KUKA KRL program: f1_Kuka_APT207T02S07.SRC

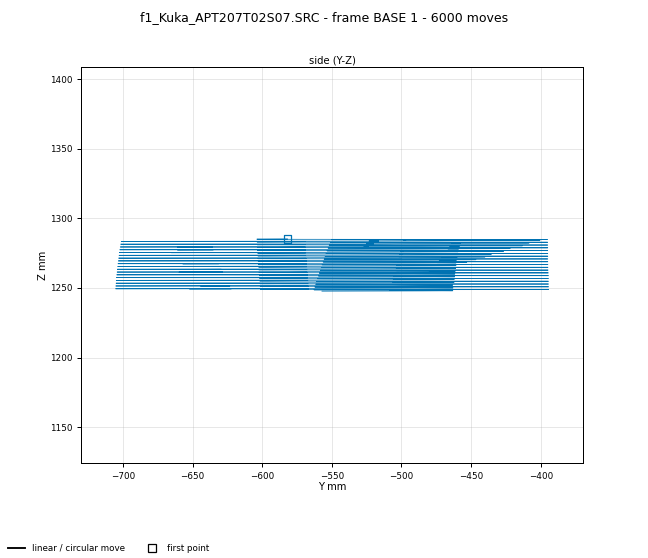
[picture p0: tool path of f1_Kuka_APT207T02S07.SRC in frame BASE 1, 6000 of 6001 moves have a stored position in this frame; points joined in program order, loops and branches not executed]
&ACCESS RVP
&REL 2
&PARAM TEMPLATE = C:\KRC\Roboter\Template\vorgabe
&PARAM EDITMASK = *
DEF f1_Kuka_APT207T02S07()


;FOLD INI;%{PE}%V3.2.0,%MKUKATPBASIS,%CINIT,%VCOMMON,%P
  ;FOLD BAS INI;%{E}%V3.2.0,%MKUKATPBASIS,%CINIT,%VINIT,%P
    GLOBAL INTERRUPT DECL 3 WHEN $STOPMESS==TRUE DO IR_STOPM ( )
    INTERRUPT ON 3
    BAS (#INITMOV,0 )
  ;ENDFOLD (BAS INI)
  ;FOLD USER INI;%{E}%V3.2.0,%MKUKATPUSER,%CINIT,%VINIT,%P
    ;Make your modifications here
  ;ENDFOLD (USER INI)
;ENDFOLD (INI)


;*** Make Null PTP Move
  PTP $pos_act

;*** Auto Load The Correct TOOL Data
  $tool=tool_data[2]

;*** Auto Load The Correct BASE Data
  $base=base_data[1]

  $ADVANCE = 5

;*** Restate Last Velocity
MMPM(30000.0)
SetRPM(8000)
LIN {X 0.048,Y -581.826,Z 1285.220,A 0.000,B 0.000,C 90.000,E1 75.589} C_DIS
LIN {X -0.200,Y -582.772,Z 1285.213,A 0.000,B 0.000,C 90.000,E1 74.267} C_DIS
LIN {X 0.309,Y -583.459,Z 1285.207,A 0.000,B 0.000,C 90.000,E1 73.142} C_DIS
LIN {X 0.170,Y -584.748,Z 1285.196,A 0.000,B 0.000,C 90.000,E1 71.275} C_DIS
LIN {X 0.250,Y -585.720,Z 1285.186,A 0.000,B 0.000,C 90.000,E1 69.390} C_DIS
LIN {X 0.080,Y -587.159,Z 1285.172,A 0.000,B 0.000,C 90.000,E1 66.997} C_DIS
LIN {X -0.086,Y -588.355,Z 1285.163,A 0.000,B 0.000,C 90.000,E1 65.409} C_DIS
LIN {X 0.318,Y -589.579,Z 1285.155,A 0.000,B 0.000,C 90.000,E1 63.768} C_DIS
LIN {X -0.318,Y -590.924,Z 1285.146,A 0.000,B 0.000,C 90.000,E1 62.231} C_DIS
LIN {X 0.047,Y -592.714,Z 1285.135,A 0.000,B 0.000,C 90.000,E1 60.333} C_DIS
LIN {X 0.246,Y -594.610,Z 1285.125,A 0.000,B 0.000,C 90.000,E1 58.456} C_DIS
LIN {X -0.011,Y -596.580,Z 1285.115,A 0.000,B 0.000,C 90.000,E1 56.628} C_DIS
LIN {X -0.137,Y -598.137,Z 1285.106,A 0.000,B 0.000,C 90.000,E1 55.055} C_DIS
LIN {X -0.029,Y -599.606,Z 1285.097,A 0.000,B 0.000,C 90.000,E1 53.463} C_DIS
LIN {X -0.243,Y -600.936,Z 1285.088,A 0.000,B 0.000,C 90.000,E1 51.904} C_DIS
LIN {X 0.057,Y -601.935,Z 1285.081,A 0.000,B 0.000,C 90.000,E1 50.561} C_DIS
LIN {X -0.015,Y -602.640,Z 1285.074,A 0.000,B 0.000,C 90.000,E1 49.256} C_DIS
LIN {X 0.252,Y -603.219,Z 1285.066,A 0.000,B 0.000,C 90.000,E1 47.919} C_DIS
LIN {X 0.129,Y -603.619,Z 1285.059,A 0.000,B 0.000,C 90.000,E1 46.620} C_DIS
LIN {X 0.184,Y -603.812,Z 1285.053,A 0.000,B 0.000,C 90.000,E1 45.567} C_DIS
LIN {X 0.047,Y -603.766,Z 1285.046,A 0.000,B 0.000,C 90.000,E1 44.271} C_DIS
LIN {X 0.303,Y -603.652,Z 1285.042,A 0.000,B 0.000,C 90.000,E1 43.461} C_DIS
LIN {X -0.019,Y -603.203,Z 1285.033,A 0.000,B 0.000,C 90.000,E1 41.919} C_DIS
LIN {X -0.182,Y -602.884,Z 1285.029,A 0.000,B 0.000,C 90.000,E1 41.148} C_DIS
LIN {X 0.183,Y -602.034,Z 1285.018,A 0.000,B 0.000,C 90.000,E1 39.277} C_DIS
LIN {X -0.130,Y -601.379,Z 1285.013,A 0.000,B 0.000,C 90.000,E1 38.257} C_DIS
LIN {X -0.203,Y -600.134,Z 1285.005,A 0.000,B 0.000,C 90.000,E1 36.950} C_DIS
LIN {X 0.177,Y -598.525,Z 1284.998,A 0.000,B 0.000,C 90.000,E1 35.598} C_DIS
LIN {X 0.054,Y -597.309,Z 1284.994,A 0.000,B 0.000,C 90.000,E1 34.818} C_DIS
LIN {X -0.084,Y -595.954,Z 1284.989,A 0.000,B 0.000,C 90.000,E1 34.040} C_DIS
LIN {X 0.147,Y -593.900,Z 1284.983,A 0.000,B 0.000,C 90.000,E1 32.959} C_DIS
LIN {X 0.253,Y -592.666,Z 1284.980,A 0.000,B 0.000,C 90.000,E1 32.418} C_DIS
LIN {X -0.062,Y -589.778,Z 1284.974,A 0.000,B 0.000,C 90.000,E1 31.386} C_DIS
LIN {X 0.014,Y -588.135,Z 1284.971,A 0.000,B 0.000,C 90.000,E1 30.846} C_DIS
LIN {X -0.045,Y -585.442,Z 1284.967,A 0.000,B 0.000,C 90.000,E1 30.050} C_DIS
LIN {X 0.376,Y -582.311,Z 1284.963,A 0.000,B 0.000,C 90.000,E1 29.205} C_DIS
LIN {X 0.046,Y -579.263,Z 1284.959,A 0.000,B 0.000,C 90.000,E1 28.565} C_DIS
LIN {X -0.185,Y -574.540,Z 1284.953,A 0.000,B 0.000,C 90.000,E1 27.641} C_DIS
LIN {X -0.067,Y -570.770,Z 1284.950,A 0.000,B 0.000,C 90.000,E1 26.950} C_DIS
LIN {X 0.275,Y -566.596,Z 1284.946,A 0.000,B 0.000,C 90.000,E1 26.232} C_DIS
LIN {X -0.088,Y -563.016,Z 1284.943,A 0.000,B 0.000,C 90.000,E1 25.720} C_DIS
LIN {X -0.067,Y -558.285,Z 1284.939,A 0.000,B 0.000,C 90.000,E1 25.027} C_DIS
LIN {X -0.011,Y -553.284,Z 1284.935,A 0.000,B 0.000,C 90.000,E1 24.335} C_DIS
LIN {X 0.041,Y -548.855,Z 1284.932,A 0.000,B 0.000,C 90.000,E1 23.770} C_DIS
LIN {X 0.218,Y -540.504,Z 1284.927,A 0.000,B 0.000,C 90.000,E1 22.770} C_DIS
LIN {X 0.093,Y -534.167,Z 1284.923,A 0.000,B 0.000,C 90.000,E1 22.078} C_DIS
LIN {X 0.176,Y -526.388,Z 1284.918,A 0.000,B 0.000,C 90.000,E1 21.227} C_DIS
LIN {X 0.260,Y -515.939,Z 1284.912,A 0.000,B 0.000,C 90.000,E1 20.120} C_DIS
LIN {X 0.127,Y -503.629,Z 1284.905,A 0.000,B 0.000,C 90.000,E1 18.906} C_DIS
LIN {X -0.214,Y -493.980,Z 1284.900,A 0.000,B 0.000,C 90.000,E1 18.000} C_DIS
LIN {X 0.123,Y -485.479,Z 1284.896,A 0.000,B 0.000,C 90.000,E1 17.166} C_DIS
LIN {X -0.200,Y -477.046,Z 1284.891,A 0.000,B 0.000,C 90.000,E1 16.441} C_DIS
LIN {X 0.098,Y -466.700,Z 1284.886,A 0.000,B 0.000,C 90.000,E1 15.481} C_DIS
LIN {X 0.071,Y -446.110,Z 1284.876,A 0.000,B 0.000,C 90.000,E1 13.592} C_DIS
LIN {X -0.108,Y -422.917,Z 1284.863,A 0.000,B 0.000,C 90.000,E1 11.299} C_DIS
LIN {X -0.089,Y -405.684,Z 1284.852,A 0.000,B 0.000,C 90.000,E1 9.434} C_DIS
LIN {X -0.183,Y -400.098,Z 1284.849,A 0.000,B 0.000,C 90.000,E1 8.803} C_DIS
LIN {X 0.108,Y -396.550,Z 1284.846,A 0.000,B 0.000,C 90.000,E1 8.276} C_DIS
LIN {X -0.073,Y -395.161,Z 1284.845,A 0.000,B 0.000,C 90.000,E1 8.049} C_DIS
LIN {X -0.110,Y -395.161,Z 1284.845,A 0.000,B 0.000,C 90.000,E1 8.049} C_DIS
LIN {X 0.067,Y -395.273,Z 1284.844,A 0.000,B 0.000,C 90.000,E1 7.936} C_DIS
LIN {X 0.028,Y -395.301,Z 1284.844,A 0.000,B 0.000,C 90.000,E1 7.936} C_DIS
LIN {X 0.134,Y -395.933,Z 1284.844,A 0.000,B 0.000,C 90.000,E1 7.814} C_DIS
LIN {X 0.006,Y -399.237,Z 1284.842,A 0.000,B 0.000,C 90.000,E1 7.530} C_DIS
LIN {X 0.124,Y -403.414,Z 1284.840,A 0.000,B 0.000,C 90.000,E1 7.239} C_DIS
LIN {X 0.177,Y -410.405,Z 1284.838,A 0.000,B 0.000,C 90.000,E1 6.834} C_DIS
LIN {X 0.174,Y -416.754,Z 1284.836,A 0.000,B 0.000,C 90.000,E1 6.429} C_DIS
LIN {X -0.121,Y -423.072,Z 1284.833,A 0.000,B 0.000,C 90.000,E1 6.024} C_DIS
LIN {X -0.122,Y -430.624,Z 1284.830,A 0.000,B 0.000,C 90.000,E1 5.448} C_DIS
LIN {X -0.194,Y -441.583,Z 1284.825,A 0.000,B 0.000,C 90.000,E1 4.588} C_DIS
LIN {X -0.037,Y -452.155,Z 1284.820,A 0.000,B 0.000,C 90.000,E1 3.669} C_DIS
LIN {X 0.164,Y -459.533,Z 1284.817,A 0.000,B 0.000,C 90.000,E1 2.980} C_DIS
LIN {X 0.220,Y -466.501,Z 1284.813,A 0.000,B 0.000,C 90.000,E1 2.293} C_DIS
LIN {X -0.131,Y -473.329,Z 1284.809,A 0.000,B 0.000,C 90.000,E1 1.604} C_DIS
LIN {X 0.114,Y -478.651,Z 1284.806,A 0.000,B 0.000,C 90.000,E1 0.974} C_DIS
LIN {X -0.058,Y -484.810,Z 1284.801,A 0.000,B 0.000,C 90.000,E1 0.229} C_DIS
LIN {X 0.015,Y -490.312,Z 1284.797,A 0.000,B 0.000,C 90.000,E1 359.484} C_DIS
LIN {X 0.044,Y -496.441,Z 1284.792,A 0.000,B 0.000,C 90.000,E1 358.568} C_DIS
LIN {X -0.029,Y -501.231,Z 1284.788,A 0.000,B 0.000,C 90.000,E1 357.822} C_DIS
LIN {X 0.231,Y -504.859,Z 1284.785,A 0.000,B 0.000,C 90.000,E1 357.192} C_DIS
LIN {X 0.241,Y -509.077,Z 1284.780,A 0.000,B 0.000,C 90.000,E1 356.445} C_DIS
LIN {X -0.218,Y -513.021,Z 1284.776,A 0.000,B 0.000,C 90.000,E1 355.755} C_DIS
LIN {X -0.210,Y -518.124,Z 1284.771,A 0.000,B 0.000,C 90.000,E1 354.723} C_DIS
LIN {X -0.090,Y -522.655,Z 1284.765,A 0.000,B 0.000,C 90.000,E1 353.685} C_DIS
LIN {X 0.087,Y -526.892,Z 1284.759,A 0.000,B 0.000,C 90.000,E1 352.648} C_DIS
LIN {X 0.101,Y -531.063,Z 1284.753,A 0.000,B 0.000,C 90.000,E1 351.489} C_DIS
LIN {X 0.130,Y -533.929,Z 1284.748,A 0.000,B 0.000,C 90.000,E1 350.622} C_DIS
LIN {X -0.250,Y -536.492,Z 1284.743,A 0.000,B 0.000,C 90.000,E1 349.803} C_DIS
LIN {X -0.069,Y -538.784,Z 1284.739,A 0.000,B 0.000,C 90.000,E1 348.926} C_DIS
LIN {X 0.214,Y -541.529,Z 1284.732,A 0.000,B 0.000,C 90.000,E1 347.757} C_DIS
LIN {X 0.003,Y -543.947,Z 1284.726,A 0.000,B 0.000,C 90.000,E1 346.645} C_DIS
LIN {X 0.172,Y -545.083,Z 1284.723,A 0.000,B 0.000,C 90.000,E1 346.061} C_DIS
LIN {X 0.131,Y -546.942,Z 1284.716,A 0.000,B 0.000,C 90.000,E1 344.936} C_DIS
LIN {X 0.021,Y -548.089,Z 1284.712,A 0.000,B 0.000,C 90.000,E1 344.102} C_DIS
LIN {X -0.075,Y -548.968,Z 1284.707,A 0.000,B 0.000,C 90.000,E1 343.268} C_DIS
LIN {X 0.091,Y -549.899,Z 1284.701,A 0.000,B 0.000,C 90.000,E1 342.127} C_DIS
LIN {X 0.182,Y -550.312,Z 1284.696,A 0.000,B 0.000,C 90.000,E1 341.275} C_DIS
LIN {X 0.280,Y -550.335,Z 1284.691,A 0.000,B 0.000,C 90.000,E1 340.423} C_DIS
LIN {X -0.136,Y -550.059,Z 1284.687,A 0.000,B 0.000,C 90.000,E1 339.625} C_DIS
LIN {X 0.206,Y -549.736,Z 1284.684,A 0.000,B 0.000,C 90.000,E1 339.028} C_DIS
LIN {X 0.227,Y -549.232,Z 1284.681,A 0.000,B 0.000,C 90.000,E1 338.465} C_DIS
LIN {X -0.202,Y -548.198,Z 1284.676,A 0.000,B 0.000,C 90.000,E1 337.667} C_DIS
LIN {X 0.074,Y -546.828,Z 1284.671,A 0.000,B 0.000,C 90.000,E1 336.794} C_DIS
LIN {X -0.164,Y -545.362,Z 1284.667,A 0.000,B 0.000,C 90.000,E1 335.973} C_DIS
LIN {X -0.165,Y -544.289,Z 1284.663,A 0.000,B 0.000,C 90.000,E1 335.409} C_DIS
LIN {X 0.086,Y -542.056,Z 1284.659,A 0.000,B 0.000,C 90.000,E1 334.537} C_DIS
LIN {X 0.033,Y -539.633,Z 1284.654,A 0.000,B 0.000,C 90.000,E1 333.691} C_DIS
LIN {X -0.283,Y -536.936,Z 1284.649,A 0.000,B 0.000,C 90.000,E1 332.871} C_DIS
LIN {X 0.089,Y -533.883,Z 1284.644,A 0.000,B 0.000,C 90.000,E1 331.975} C_DIS
LIN {X 0.243,Y -531.727,Z 1284.641,A 0.000,B 0.000,C 90.000,E1 331.385} C_DIS
LIN {X 0.231,Y -528.707,Z 1284.637,A 0.000,B 0.000,C 90.000,E1 330.667} C_DIS
LIN {X 0.293,Y -524.436,Z 1284.632,A 0.000,B 0.000,C 90.000,E1 329.793} C_DIS
LIN {X -0.076,Y -521.409,Z 1284.629,A 0.000,B 0.000,C 90.000,E1 329.253} C_DIS
LIN {X -0.168,Y -508.672,Z 1284.616,A 0.000,B 0.000,C 90.000,E1 326.914} C_DIS
LIN {X -0.044,Y -504.398,Z 1284.611,A 0.000,B 0.000,C 90.000,E1 326.008} C_DIS
LIN {X -0.108,Y -501.931,Z 1284.607,A 0.000,B 0.000,C 90.000,E1 325.308} C_DIS
LIN {X 0.189,Y -501.065,Z 1284.606,A 0.000,B 0.000,C 90.000,E1 324.975} C_DIS
LIN {X -0.063,Y -499.234,Z 1284.601,A 0.000,B 0.000,C 90.000,E1 324.116} C_DIS
LIN {X -0.038,Y -497.969,Z 1284.596,A 0.000,B 0.000,C 90.000,E1 323.210} C_DIS
LIN {X 0.136,Y -497.147,Z 1284.589,A 0.000,B 0.000,C 90.000,E1 321.984} C_DIS
LIN {X -0.229,Y -496.725,Z 1284.581,A 0.000,B 0.000,C 90.000,E1 320.517} C_DIS
LIN {X 0.043,Y -496.935,Z 1284.572,A 0.000,B 0.000,C 90.000,E1 318.976} C_DIS
LIN {X 0.039,Y -497.249,Z 1284.560,A 0.000,B 0.000,C 90.000,E1 316.863} C_DIS
LIN {X -0.207,Y -497.490,Z 1284.550,A 0.000,B 0.000,C 90.000,E1 315.081} C_DIS
LIN {X -0.203,Y -497.954,Z 1284.535,A 0.000,B 0.000,C 90.000,E1 312.366} C_DIS
LIN {X 0.091,Y -498.258,Z 1284.527,A 0.000,B 0.000,C 90.000,E1 310.825} C_DIS
LIN {X -0.122,Y -498.440,Z 1284.520,A 0.000,B 0.000,C 90.000,E1 309.644} C_DIS
LIN {X -0.199,Y -498.339,Z 1284.515,A 0.000,B 0.000,C 90.000,E1 308.749} C_DIS
LIN {X 0.112,Y -497.903,Z 1284.510,A 0.000,B 0.000,C 90.000,E1 307.810} C_DIS
LIN {X -0.148,Y -497.351,Z 1284.507,A 0.000,B 0.000,C 90.000,E1 307.237} C_DIS
LIN {X 0.284,Y -496.489,Z 1284.503,A 0.000,B 0.000,C 90.000,E1 306.583} C_DIS
LIN {X 0.151,Y -495.889,Z 1284.502,A 0.000,B 0.000,C 90.000,E1 306.297} C_DIS
LIN {X 0.015,Y -495.108,Z 1284.500,A 0.000,B 0.000,C 90.000,E1 306.011} C_DIS
LIN {X -0.122,Y -493.974,Z 1284.498,A 0.000,B 0.000,C 90.000,E1 305.724} C_DIS
LIN {X 0.004,Y -476.992,Z 1284.482,A 0.000,B 0.000,C 90.000,E1 302.801} C_DIS
LIN {X -0.163,Y -462.651,Z 1284.467,A 0.000,B 0.000,C 90.000,E1 300.001} C_DIS
LIN {X -0.075,Y -449.320,Z 1284.450,A 0.000,B 0.000,C 90.000,E1 296.950} C_DIS
LIN {X 0.022,Y -438.317,Z 1284.433,A 0.000,B 0.000,C 90.000,E1 294.003} C_DIS
LIN {X 0.060,Y -427.853,Z 1284.415,A 0.000,B 0.000,C 90.000,E1 290.684} C_DIS
LIN {X 0.007,Y -418.374,Z 1284.394,A 0.000,B 0.000,C 90.000,E1 286.985} C_DIS
LIN {X 0.007,Y -410.353,Z 1284.372,A 0.000,B 0.000,C 90.000,E1 282.883} C_DIS
LIN {X 0.108,Y -405.581,Z 1284.353,A 0.000,B 0.000,C 90.000,E1 279.500} C_DIS
LIN {X -0.078,Y -405.689,Z 1284.333,A 0.000,B 0.000,C 90.000,E1 275.967} C_DIS
LIN {X -0.040,Y -403.463,Z 1284.304,A 0.000,B 0.000,C 90.000,E1 270.745} C_DIS
LIN {X -0.073,Y -403.247,Z 1284.302,A 0.000,B 0.000,C 90.000,E1 270.401} C_DIS
LIN {X 0.093,Y -400.475,Z 1284.286,A 0.000,B 0.000,C 90.000,E1 267.421} C_DIS
LIN {X 0.055,Y -400.476,Z 1284.286,A 0.000,B 0.000,C 90.000,E1 267.421} C_DIS
LIN {X -0.055,Y -405.330,Z 1284.250,A 0.000,B 0.000,C 90.000,E1 260.971} C_DIS
LIN {X 0.004,Y -411.969,Z 1284.225,A 0.000,B 0.000,C 90.000,E1 256.464} C_DIS
LIN {X -0.169,Y -419.748,Z 1284.204,A 0.000,B 0.000,C 90.000,E1 252.725} C_DIS
LIN {X -0.092,Y -428.611,Z 1284.185,A 0.000,B 0.000,C 90.000,E1 249.337} C_DIS
LIN {X 0.007,Y -439.259,Z 1284.167,A 0.000,B 0.000,C 90.000,E1 245.997} C_DIS
LIN {X 0.176,Y -451.103,Z 1284.149,A 0.000,B 0.000,C 90.000,E1 242.871} C_DIS
LIN {X 0.067,Y -460.165,Z 1284.138,A 0.000,B 0.000,C 90.000,E1 240.795} C_DIS
LIN {X 0.188,Y -461.036,Z 1284.136,A 0.000,B 0.000,C 90.000,E1 240.461} C_DIS
LIN {X -0.088,Y -461.611,Z 1284.134,A 0.000,B 0.000,C 90.000,E1 240.177} C_DIS
LIN {X -0.062,Y -462.296,Z 1284.131,A 0.000,B 0.000,C 90.000,E1 239.537} C_DIS
LIN {X 0.203,Y -462.605,Z 1284.127,A 0.000,B 0.000,C 90.000,E1 238.869} C_DIS
LIN {X -0.033,Y -462.663,Z 1284.122,A 0.000,B 0.000,C 90.000,E1 237.946} C_DIS
LIN {X -0.027,Y -462.349,Z 1284.117,A 0.000,B 0.000,C 90.000,E1 236.993} C_DIS
LIN {X -0.021,Y -461.709,Z 1284.110,A 0.000,B 0.000,C 90.000,E1 235.722} C_DIS
LIN {X -0.015,Y -460.306,Z 1284.095,A 0.000,B 0.000,C 90.000,E1 233.176} C_DIS
LIN {X 0.090,Y -459.422,Z 1284.085,A 0.000,B 0.000,C 90.000,E1 231.251} C_DIS
LIN {X 0.149,Y -458.484,Z 1284.071,A 0.000,B 0.000,C 90.000,E1 228.690} C_DIS
LIN {X 0.108,Y -457.814,Z 1284.058,A 0.000,B 0.000,C 90.000,E1 226.458} C_DIS
LIN {X -0.268,Y -457.345,Z 1284.044,A 0.000,B 0.000,C 90.000,E1 223.947} C_DIS
LIN {X 0.127,Y -457.909,Z 1284.024,A 0.000,B 0.000,C 90.000,E1 220.378} C_DIS
LIN {X -0.164,Y -458.661,Z 1284.012,A 0.000,B 0.000,C 90.000,E1 218.177} C_DIS
LIN {X 0.145,Y -463.330,Z 1283.978,A 0.000,B 0.000,C 90.000,E1 212.084} C_DIS
LIN {X 0.099,Y -466.009,Z 1283.966,A 0.000,B 0.000,C 90.000,E1 209.873} C_DIS
LIN {X -0.040,Y -469.420,Z 1283.950,A 0.000,B 0.000,C 90.000,E1 207.052} C_DIS
LIN {X 0.108,Y -471.545,Z 1283.942,A 0.000,B 0.000,C 90.000,E1 205.463} C_DIS
LIN {X 0.074,Y -474.369,Z 1283.931,A 0.000,B 0.000,C 90.000,E1 203.590} C_DIS
LIN {X 0.051,Y -478.675,Z 1283.916,A 0.000,B 0.000,C 90.000,E1 200.791} C_DIS
LIN {X 0.112,Y -482.749,Z 1283.902,A 0.000,B 0.000,C 90.000,E1 198.308} C_DIS
LIN {X -0.183,Y -485.961,Z 1283.892,A 0.000,B 0.000,C 90.000,E1 196.496} C_DIS
LIN {X -0.096,Y -488.690,Z 1283.883,A 0.000,B 0.000,C 90.000,E1 194.954} C_DIS
LIN {X 0.042,Y -491.381,Z 1283.875,A 0.000,B 0.000,C 90.000,E1 193.411} C_DIS
LIN {X 0.111,Y -494.109,Z 1283.866,A 0.000,B 0.000,C 90.000,E1 191.883} C_DIS
LIN {X 0.129,Y -496.849,Z 1283.858,A 0.000,B 0.000,C 90.000,E1 190.366} C_DIS
LIN {X -0.044,Y -500.740,Z 1283.846,A 0.000,B 0.000,C 90.000,E1 188.276} C_DIS
LIN {X 0.155,Y -502.380,Z 1283.841,A 0.000,B 0.000,C 90.000,E1 187.352} C_DIS
LIN {X -0.253,Y -504.575,Z 1283.834,A 0.000,B 0.000,C 90.000,E1 186.201} C_DIS
LIN {X -0.192,Y -507.140,Z 1283.826,A 0.000,B 0.000,C 90.000,E1 184.702} C_DIS
LIN {X -0.162,Y -509.747,Z 1283.818,A 0.000,B 0.000,C 90.000,E1 183.212} C_DIS
LIN {X -0.057,Y -512.196,Z 1283.810,A 0.000,B 0.000,C 90.000,E1 181.718} C_DIS
LIN {X 0.134,Y -514.028,Z 1283.803,A 0.000,B 0.000,C 90.000,E1 180.516} C_DIS
LIN {X -0.089,Y -515.367,Z 1283.798,A 0.000,B 0.000,C 90.000,E1 179.656} C_DIS
LIN {X 0.101,Y -517.474,Z 1283.790,A 0.000,B 0.000,C 90.000,E1 178.165} C_DIS
LIN {X -0.152,Y -518.982,Z 1283.783,A 0.000,B 0.000,C 90.000,E1 177.020} C_DIS
LIN {X 0.190,Y -520.307,Z 1283.777,A 0.000,B 0.000,C 90.000,E1 175.812} C_DIS
LIN {X -0.019,Y -521.600,Z 1283.769,A 0.000,B 0.000,C 90.000,E1 174.375} C_DIS
LIN {X -0.152,Y -522.343,Z 1283.762,A 0.000,B 0.000,C 90.000,E1 173.223} C_DIS
LIN {X -0.280,Y -523.033,Z 1283.754,A 0.000,B 0.000,C 90.000,E1 171.781} C_DIS
LIN {X 0.183,Y -523.263,Z 1283.748,A 0.000,B 0.000,C 90.000,E1 170.566} C_DIS
LIN {X 0.231,Y -523.185,Z 1283.740,A 0.000,B 0.000,C 90.000,E1 169.106} C_DIS
LIN {X -0.230,Y -522.561,Z 1283.732,A 0.000,B 0.000,C 90.000,E1 167.701} C_DIS
LIN {X -0.083,Y -521.708,Z 1283.725,A 0.000,B 0.000,C 90.000,E1 166.520} C_DIS
LIN {X 0.055,Y -520.793,Z 1283.719,A 0.000,B 0.000,C 90.000,E1 165.338} C_DIS
LIN {X -0.201,Y -519.262,Z 1283.709,A 0.000,B 0.000,C 90.000,E1 163.614} C_DIS
LIN {X 0.118,Y -517.420,Z 1283.698,A 0.000,B 0.000,C 90.000,E1 161.529} C_DIS
LIN {X -0.141,Y -516.682,Z 1283.693,A 0.000,B 0.000,C 90.000,E1 160.678} C_DIS
LIN {X -0.141,Y -516.324,Z 1283.684,A 0.000,B 0.000,C 90.000,E1 159.209} C_DIS
LIN {X 0.259,Y -516.711,Z 1283.680,A 0.000,B 0.000,C 90.000,E1 158.284} C_DIS
LIN {X 0.324,Y -517.764,Z 1283.673,A 0.000,B 0.000,C 90.000,E1 157.102} C_DIS
LIN {X 0.124,Y -518.879,Z 1283.670,A 0.000,B 0.000,C 90.000,E1 156.538} C_DIS
LIN {X -0.068,Y -520.301,Z 1283.667,A 0.000,B 0.000,C 90.000,E1 155.973} C_DIS
LIN {X 0.224,Y -522.225,Z 1283.663,A 0.000,B 0.000,C 90.000,E1 155.357} C_DIS
LIN {X 0.053,Y -524.712,Z 1283.660,A 0.000,B 0.000,C 90.000,E1 154.793} C_DIS
LIN {X -0.025,Y -528.710,Z 1283.656,A 0.000,B 0.000,C 90.000,E1 154.076} C_DIS
LIN {X -0.003,Y -531.578,Z 1283.654,A 0.000,B 0.000,C 90.000,E1 153.640} C_DIS
LIN {X -0.089,Y -539.433,Z 1283.648,A 0.000,B 0.000,C 90.000,E1 152.666} C_DIS
LIN {X 0.271,Y -548.357,Z 1283.643,A 0.000,B 0.000,C 90.000,E1 151.641} C_DIS
LIN {X 0.153,Y -565.525,Z 1283.633,A 0.000,B 0.000,C 90.000,E1 149.999} C_DIS
LIN {X -0.047,Y -574.734,Z 1283.629,A 0.000,B 0.000,C 90.000,E1 149.154} C_DIS
LIN {X -0.057,Y -581.132,Z 1283.625,A 0.000,B 0.000,C 90.000,E1 148.535} C_DIS
LIN {X -0.226,Y -589.974,Z 1283.620,A 0.000,B 0.000,C 90.000,E1 147.661} C_DIS
LIN {X -0.070,Y -596.134,Z 1283.617,A 0.000,B 0.000,C 90.000,E1 146.993} C_DIS
LIN {X -0.164,Y -601.805,Z 1283.613,A 0.000,B 0.000,C 90.000,E1 146.342} C_DIS
LIN {X -0.005,Y -606.058,Z 1283.610,A 0.000,B 0.000,C 90.000,E1 145.801} C_DIS
LIN {X 0.182,Y -610.024,Z 1283.607,A 0.000,B 0.000,C 90.000,E1 145.261} C_DIS
LIN {X 0.218,Y -614.724,Z 1283.604,A 0.000,B 0.000,C 90.000,E1 144.609} C_DIS
LIN {X -0.038,Y -618.124,Z 1283.601,A 0.000,B 0.000,C 90.000,E1 144.116} C_DIS
LIN {X 0.050,Y -622.762,Z 1283.596,A 0.000,B 0.000,C 90.000,E1 143.336} C_DIS
LIN {X -0.158,Y -625.657,Z 1283.594,A 0.000,B 0.000,C 90.000,E1 142.844} C_DIS
LIN {X 0.165,Y -627.743,Z 1283.591,A 0.000,B 0.000,C 90.000,E1 142.431} C_DIS
LIN {X 0.125,Y -633.916,Z 1283.584,A 0.000,B 0.000,C 90.000,E1 141.170} C_DIS
LIN {X -0.247,Y -638.218,Z 1283.579,A 0.000,B 0.000,C 90.000,E1 140.194} C_DIS
LIN {X -0.079,Y -642.231,Z 1283.573,A 0.000,B 0.000,C 90.000,E1 139.175} C_DIS
LIN {X 0.002,Y -646.873,Z 1283.566,A 0.000,B 0.000,C 90.000,E1 137.919} C_DIS
LIN {X 0.227,Y -650.332,Z 1283.561,A 0.000,B 0.000,C 90.000,E1 136.905} C_DIS
LIN {X -0.003,Y -654.618,Z 1283.554,A 0.000,B 0.000,C 90.000,E1 135.688} C_DIS
LIN {X 0.231,Y -660.564,Z 1283.544,A 0.000,B 0.000,C 90.000,E1 133.947} C_DIS
LIN {X -0.309,Y -664.882,Z 1283.537,A 0.000,B 0.000,C 90.000,E1 132.771} C_DIS
LIN {X 0.155,Y -669.089,Z 1283.531,A 0.000,B 0.000,C 90.000,E1 131.515} C_DIS
LIN {X -0.184,Y -673.808,Z 1283.523,A 0.000,B 0.000,C 90.000,E1 130.092} C_DIS
LIN {X -0.029,Y -677.602,Z 1283.516,A 0.000,B 0.000,C 90.000,E1 128.874} C_DIS
LIN {X -0.290,Y -679.747,Z 1283.512,A 0.000,B 0.000,C 90.000,E1 128.177} C_DIS
LIN {X 0.070,Y -683.148,Z 1283.505,A 0.000,B 0.000,C 90.000,E1 126.950} C_DIS
LIN {X 0.082,Y -686.305,Z 1283.499,A 0.000,B 0.000,C 90.000,E1 125.758} C_DIS
LIN {X -0.418,Y -689.158,Z 1283.492,A 0.000,B 0.000,C 90.000,E1 124.612} C_DIS
LIN {X 0.041,Y -691.302,Z 1283.487,A 0.000,B 0.000,C 90.000,E1 123.627} C_DIS
LIN {X 0.122,Y -692.680,Z 1283.483,A 0.000,B 0.000,C 90.000,E1 122.911} C_DIS
LIN {X -0.338,Y -694.452,Z 1283.478,A 0.000,B 0.000,C 90.000,E1 122.005} C_DIS
LIN {X 0.048,Y -696.407,Z 1283.471,A 0.000,B 0.000,C 90.000,E1 120.797} C_DIS
LIN {X -0.144,Y -697.875,Z 1283.466,A 0.000,B 0.000,C 90.000,E1 119.873} C_DIS
LIN {X -0.052,Y -699.481,Z 1283.459,A 0.000,B 0.000,C 90.000,E1 118.693} C_DIS
LIN {X -0.210,Y -700.493,Z 1283.454,A 0.000,B 0.000,C 90.000,E1 117.769} C_DIS
LIN {X -0.017,Y -701.034,Z 1283.450,A 0.000,B 0.000,C 90.000,E1 117.052} C_DIS
LIN {X 0.140,Y -701.210,Z 1283.445,A 0.000,B 0.000,C 90.000,E1 116.104} C_DIS
LIN {X -0.215,Y -701.232,Z 1283.444,A 0.000,B 0.000,C 90.000,E1 115.899} C_DIS
LIN {X 0.306,Y -700.865,Z 1283.440,A 0.000,B 0.000,C 90.000,E1 115.155} C_DIS
LIN {X -0.077,Y -700.397,Z 1283.437,A 0.000,B 0.000,C 90.000,E1 114.719} C_DIS
LIN {X -0.171,Y -699.673,Z 1283.435,A 0.000,B 0.000,C 90.000,E1 114.259} C_DIS
LIN {X -0.189,Y -699.008,Z 1283.433,A 0.000,B 0.000,C 90.000,E1 114.027} C_DIS
LIN {X 0.342,Y -697.245,Z 1283.431,A 0.000,B 0.000,C 90.000,E1 113.515} C_DIS
LIN {X -0.168,Y -696.536,Z 1283.430,A 0.000,B 0.000,C 90.000,E1 113.439} C_DIS
LIN {X 0.062,Y -693.012,Z 1283.428,A 0.000,B 0.000,C 90.000,E1 112.950} C_DIS
LIN {X 0.185,Y -691.812,Z 1283.427,A 0.000,B 0.000,C 90.000,E1 112.823} C_DIS
LIN {X 0.051,Y -689.979,Z 1283.426,A 0.000,B 0.000,C 90.000,E1 112.717} C_DIS
LIN {X 0.346,Y -683.033,Z 1283.424,A 0.000,B 0.000,C 90.000,E1 112.333} C_DIS
LIN {X 0.207,Y -678.619,Z 1283.423,A 0.000,B 0.000,C 90.000,E1 112.206} C_DIS
LIN {X 0.175,Y -669.996,Z 1283.423,A 0.000,B 0.000,C 90.000,E1 112.078} C_DIS
LIN {X 0.038,Y -667.165,Z 1283.423,A 0.000,B 0.000,C 90.000,E1 112.078} C_DIS
LIN {X -0.030,Y -662.781,Z 1283.423,A 0.000,B 0.000,C 90.000,E1 112.078} C_DIS
LIN {X -0.095,Y -640.134,Z 1283.423,A 0.000,B 0.000,C 90.000,E1 112.078} C_DIS
LIN {X 0.101,Y -638.371,Z 1283.422,A 0.000,B 0.000,C 90.000,E1 112.025} C_DIS
LIN {X -0.010,Y -636.764,Z 1283.422,A 0.000,B 0.000,C 90.000,E1 111.972} C_DIS
LIN {X -0.056,Y -636.749,Z 1283.422,A 0.000,B 0.000,C 90.000,E1 111.972} C_DIS
LIN {X 0.329,Y -637.495,Z 1283.421,A 0.000,B 0.000,C 90.000,E1 111.716} C_DIS
LIN {X 0.116,Y -639.891,Z 1283.419,A 0.000,B 0.000,C 90.000,E1 111.354} C_DIS
LIN {X 0.072,Y -646.351,Z 1283.414,A 0.000,B 0.000,C 90.000,E1 110.482} C_DIS
LIN {X -0.021,Y -649.800,Z 1283.411,A 0.000,B 0.000,C 90.000,E1 109.993} C_DIS
LIN {X -0.270,Y -653.548,Z 1283.408,A 0.000,B 0.000,C 90.000,E1 109.396} C_DIS
LIN {X -0.274,Y -656.849,Z 1283.404,A 0.000,B 0.000,C 90.000,E1 108.779} C_DIS
LIN {X 0.207,Y -660.355,Z 1283.400,A 0.000,B 0.000,C 90.000,E1 108.000} C_DIS
LIN {X 0.097,Y -663.582,Z 1283.396,A 0.000,B 0.000,C 90.000,E1 107.275} C_DIS
LIN {X 0.012,Y -666.414,Z 1283.392,A 0.000,B 0.000,C 90.000,E1 106.551} C_DIS
LIN {X -0.235,Y -668.763,Z 1283.388,A 0.000,B 0.000,C 90.000,E1 105.843} C_DIS
LIN {X -0.384,Y -670.183,Z 1283.385,A 0.000,B 0.000,C 90.000,E1 105.371} C_DIS
LIN {X 0.233,Y -671.858,Z 1283.381,A 0.000,B 0.000,C 90.000,E1 104.592} C_DIS
LIN {X 0.106,Y -672.776,Z 1283.379,A 0.000,B 0.000,C 90.000,E1 104.120} C_DIS
LIN {X -0.016,Y -673.524,Z 1283.376,A 0.000,B 0.000,C 90.000,E1 103.647} C_DIS
LIN {X -0.133,Y -674.074,Z 1283.373,A 0.000,B 0.000,C 90.000,E1 103.175} C_DIS
LIN {X -0.248,Y -674.480,Z 1283.370,A 0.000,B 0.000,C 90.000,E1 102.703} C_DIS
LIN {X 0.100,Y -674.674,Z 1283.366,A 0.000,B 0.000,C 90.000,E1 101.951} C_DIS
LIN {X -0.011,Y -674.608,Z 1283.364,A 0.000,B 0.000,C 90.000,E1 101.478} C_DIS
LIN {X -0.311,Y -674.055,Z 1283.360,A 0.000,B 0.000,C 90.000,E1 100.782} C_DIS
LIN {X 0.292,Y -673.833,Z 1283.359,A 0.000,B 0.000,C 90.000,E1 100.489} C_DIS
LIN {X -0.011,Y -672.650,Z 1283.354,A 0.000,B 0.000,C 90.000,E1 99.792} C_DIS
LIN {X -0.146,Y -671.630,Z 1283.352,A 0.000,B 0.000,C 90.000,E1 99.321} C_DIS
LIN {X 0.266,Y -670.250,Z 1283.349,A 0.000,B 0.000,C 90.000,E1 98.803} C_DIS
LIN {X 0.010,Y -668.501,Z 1283.346,A 0.000,B 0.000,C 90.000,E1 98.341} C_DIS
LIN {X -0.161,Y -666.465,Z 1283.344,A 0.000,B 0.000,C 90.000,E1 97.871} C_DIS
LIN {X 0.224,Y -664.720,Z 1283.342,A 0.000,B 0.000,C 90.000,E1 97.473} C_DIS
LIN {X 0.019,Y -662.173,Z 1283.339,A 0.000,B 0.000,C 90.000,E1 97.004} C_DIS
LIN {X -0.289,Y -659.289,Z 1283.336,A 0.000,B 0.000,C 90.000,E1 96.543} C_DIS
LIN {X -0.064,Y -655.148,Z 1283.333,A 0.000,B 0.000,C 90.000,E1 95.910} C_DIS
LIN {X 0.234,Y -651.516,Z 1283.330,A 0.000,B 0.000,C 90.000,E1 95.391} C_DIS
LIN {X -0.199,Y -647.580,Z 1283.327,A 0.000,B 0.000,C 90.000,E1 94.935} C_DIS
LIN {X 0.047,Y -643.232,Z 1283.325,A 0.000,B 0.000,C 90.000,E1 94.416} C_DIS
LIN {X 0.146,Y -637.283,Z 1283.321,A 0.000,B 0.000,C 90.000,E1 93.784} C_DIS
LIN {X -0.127,Y -631.220,Z 1283.318,A 0.000,B 0.000,C 90.000,E1 93.212} C_DIS
LIN {X -0.311,Y -624.742,Z 1283.315,A 0.000,B 0.000,C 90.000,E1 92.636} C_DIS
LIN {X -0.306,Y -616.597,Z 1283.311,A 0.000,B 0.000,C 90.000,E1 91.949} C_DIS
LIN {X -0.030,Y -609.351,Z 1283.308,A 0.000,B 0.000,C 90.000,E1 91.375} C_DIS
LIN {X -0.027,Y -601.459,Z 1283.305,A 0.000,B 0.000,C 90.000,E1 90.859} C_DIS
LIN {X 0.245,Y -594.976,Z 1283.303,A 0.000,B 0.000,C 90.000,E1 90.458} C_DIS
LIN {X -0.054,Y -589.839,Z 1283.301,A 0.000,B 0.000,C 90.000,E1 90.229} C_DIS
LIN {X -0.095,Y -584.328,Z 1283.300,A 0.000,B 0.000,C 90.000,E1 90.000} C_DIS
LIN {X -0.038,Y -575.829,Z 1283.298,A 0.000,B 0.000,C 90.000,E1 89.656} C_DIS
LIN {X -0.278,Y -571.756,Z 1283.297,A 0.000,B 0.000,C 90.000,E1 89.484} C_DIS
LIN {X 0.052,Y -570.075,Z 1283.296,A 0.000,B 0.000,C 90.000,E1 89.255} C_DIS
LIN {X 0.005,Y -569.451,Z 1283.295,A 0.000,B 0.000,C 90.000,E1 89.141} C_DIS
LIN {X -0.037,Y -569.149,Z 1283.294,A 0.000,B 0.000,C 90.000,E1 88.854} C_DIS
LIN {X 0.169,Y -570.073,Z 1283.285,A 0.000,B 0.000,C 90.000,E1 87.192} C_DIS
LIN {X 0.159,Y -572.082,Z 1283.272,A 0.000,B 0.000,C 90.000,E1 85.008} C_DIS
LIN {X -0.050,Y -573.853,Z 1283.263,A 0.000,B 0.000,C 90.000,E1 83.394} C_DIS
LIN {X -0.028,Y -576.070,Z 1283.253,A 0.000,B 0.000,C 90.000,E1 81.489} C_DIS
LIN {X 0.147,Y -577.349,Z 1283.247,A 0.000,B 0.000,C 90.000,E1 80.387} C_DIS
LIN {X -0.016,Y -578.726,Z 1283.239,A 0.000,B 0.000,C 90.000,E1 79.050} C_DIS
LIN {X -0.161,Y -580.413,Z 1283.229,A 0.000,B 0.000,C 90.000,E1 77.173} C_DIS
LIN {X 0.206,Y -581.762,Z 1283.220,A 0.000,B 0.000,C 90.000,E1 75.519} C_DIS
LIN {X -0.192,Y -582.693,Z 1283.212,A 0.000,B 0.000,C 90.000,E1 74.212} C_DIS
LIN {X -0.024,Y -583.541,Z 1283.205,A 0.000,B 0.000,C 90.000,E1 72.851} C_DIS
LIN {X 0.166,Y -584.660,Z 1283.196,A 0.000,B 0.000,C 90.000,E1 71.221} C_DIS
LIN {X 0.027,Y -585.456,Z 1283.187,A 0.000,B 0.000,C 90.000,E1 69.625} C_DIS
LIN {X -0.136,Y -586.872,Z 1283.173,A 0.000,B 0.000,C 90.000,E1 67.230} C_DIS
LIN {X -0.122,Y -588.272,Z 1283.163,A 0.000,B 0.000,C 90.000,E1 65.357} C_DIS
LIN {X -0.255,Y -589.513,Z 1283.154,A 0.000,B 0.000,C 90.000,E1 63.768} C_DIS
LIN {X -0.199,Y -591.101,Z 1283.144,A 0.000,B 0.000,C 90.000,E1 61.897} C_DIS
LIN {X 0.277,Y -592.660,Z 1283.135,A 0.000,B 0.000,C 90.000,E1 60.255} C_DIS
LIN {X 0.171,Y -594.564,Z 1283.125,A 0.000,B 0.000,C 90.000,E1 58.408} C_DIS
LIN {X -0.098,Y -596.539,Z 1283.114,A 0.000,B 0.000,C 90.000,E1 56.580} C_DIS
LIN {X 0.108,Y -598.089,Z 1283.105,A 0.000,B 0.000,C 90.000,E1 54.975} C_DIS
LIN {X -0.138,Y -599.560,Z 1283.097,A 0.000,B 0.000,C 90.000,E1 53.417} C_DIS
LIN {X -0.238,Y -600.641,Z 1283.089,A 0.000,B 0.000,C 90.000,E1 52.110} C_DIS
LIN {X -0.320,Y -601.682,Z 1283.082,A 0.000,B 0.000,C 90.000,E1 50.803} C_DIS
LIN {X -0.009,Y -602.424,Z 1283.075,A 0.000,B 0.000,C 90.000,E1 49.461} C_DIS
LIN {X 0.100,Y -603.106,Z 1283.066,A 0.000,B 0.000,C 90.000,E1 47.877} C_DIS
LIN {X 0.142,Y -603.449,Z 1283.060,A 0.000,B 0.000,C 90.000,E1 46.824} C_DIS
LIN {X -0.220,Y -603.681,Z 1283.054,A 0.000,B 0.000,C 90.000,E1 45.810} C_DIS
LIN {X -0.360,Y -603.683,Z 1283.047,A 0.000,B 0.000,C 90.000,E1 44.514} C_DIS
LIN {X 0.134,Y -603.497,Z 1283.041,A 0.000,B 0.000,C 90.000,E1 43.419} C_DIS
LIN {X 0.223,Y -603.065,Z 1283.033,A 0.000,B 0.000,C 90.000,E1 41.838} C_DIS
LIN {X 0.058,Y -602.737,Z 1283.028,A 0.000,B 0.000,C 90.000,E1 41.067} C_DIS
LIN {X -0.079,Y -602.131,Z 1283.021,A 0.000,B 0.000,C 90.000,E1 39.769} C_DIS
LIN {X -0.179,Y -601.721,Z 1283.017,A 0.000,B 0.000,C 90.000,E1 38.991} C_DIS
LIN {X 0.100,Y -601.202,Z 1283.012,A 0.000,B 0.000,C 90.000,E1 38.177} C_DIS
LIN {X -0.225,Y -600.260,Z 1283.006,A 0.000,B 0.000,C 90.000,E1 37.156} C_DIS
LIN {X -0.085,Y -598.990,Z 1283.000,A 0.000,B 0.000,C 90.000,E1 36.091} C_DIS
LIN {X 0.035,Y -597.563,Z 1282.995,A 0.000,B 0.000,C 90.000,E1 35.025} C_DIS
LIN {X -0.209,Y -595.688,Z 1282.989,A 0.000,B 0.000,C 90.000,E1 33.992} C_DIS
LIN {X 0.131,Y -594.206,Z 1282.984,A 0.000,B 0.000,C 90.000,E1 33.166} C_DIS
LIN {X -0.366,Y -592.397,Z 1282.980,A 0.000,B 0.000,C 90.000,E1 32.418} C_DIS
LIN {X -0.179,Y -589.469,Z 1282.974,A 0.000,B 0.000,C 90.000,E1 31.337} C_DIS
LIN {X -0.219,Y -586.928,Z 1282.970,A 0.000,B 0.000,C 90.000,E1 30.541} C_DIS
LIN {X -0.160,Y -585.072,Z 1282.967,A 0.000,B 0.000,C 90.000,E1 30.001} C_DIS
LIN {X -0.118,Y -583.006,Z 1282.964,A 0.000,B 0.000,C 90.000,E1 29.461} C_DIS
LIN {X 0.065,Y -580.105,Z 1282.960,A 0.000,B 0.000,C 90.000,E1 28.771} C_DIS
LIN {X -0.151,Y -575.415,Z 1282.955,A 0.000,B 0.000,C 90.000,E1 27.847} C_DIS
LIN {X -0.114,Y -573.234,Z 1282.952,A 0.000,B 0.000,C 90.000,E1 27.436} C_DIS
LIN {X -0.008,Y -569.372,Z 1282.949,A 0.000,B 0.000,C 90.000,E1 26.744} C_DIS
LIN {X 0.067,Y -565.155,Z 1282.945,A 0.000,B 0.000,C 90.000,E1 26.052} C_DIS
LIN {X 0.251,Y -559.601,Z 1282.940,A 0.000,B 0.000,C 90.000,E1 25.207} C_DIS
LIN {X -0.160,Y -555.622,Z 1282.937,A 0.000,B 0.000,C 90.000,E1 24.695} C_DIS
LIN {X -0.092,Y -551.384,Z 1282.934,A 0.000,B 0.000,C 90.000,E1 24.131} C_DIS
LIN {X 0.065,Y -548.012,Z 1282.932,A 0.000,B 0.000,C 90.000,E1 23.695} C_DIS
LIN {X -0.209,Y -540.975,Z 1282.927,A 0.000,B 0.000,C 90.000,E1 22.898} C_DIS
LIN {X 0.243,Y -533.569,Z 1282.923,A 0.000,B 0.000,C 90.000,E1 22.025} C_DIS
LIN {X -0.128,Y -525.839,Z 1282.918,A 0.000,B 0.000,C 90.000,E1 21.227} C_DIS
LIN {X -0.198,Y -515.189,Z 1282.912,A 0.000,B 0.000,C 90.000,E1 20.120} C_DIS
LIN {X -0.123,Y -504.164,Z 1282.906,A 0.000,B 0.000,C 90.000,E1 19.014} C_DIS
LIN {X -0.221,Y -493.016,Z 1282.900,A 0.000,B 0.000,C 90.000,E1 17.946} C_DIS
LIN {X 0.202,Y -485.843,Z 1282.896,A 0.000,B 0.000,C 90.000,E1 17.221} C_DIS
LIN {X 0.103,Y -478.474,Z 1282.892,A 0.000,B 0.000,C 90.000,E1 16.567} C_DIS
LIN {X -0.127,Y -466.637,Z 1282.886,A 0.000,B 0.000,C 90.000,E1 15.536} C_DIS
LIN {X -0.012,Y -447.492,Z 1282.877,A 0.000,B 0.000,C 90.000,E1 13.772} C_DIS
LIN {X 0.175,Y -425.689,Z 1282.865,A 0.000,B 0.000,C 90.000,E1 11.591} C_DIS
LIN {X -0.147,Y -410.043,Z 1282.855,A 0.000,B 0.000,C 90.000,E1 9.962} C_DIS
LIN {X -0.148,Y -400.244,Z 1282.849,A 0.000,B 0.000,C 90.000,E1 8.859} C_DIS
LIN {X 0.191,Y -395.967,Z 1282.846,A 0.000,B 0.000,C 90.000,E1 8.219} C_DIS
LIN {X -0.002,Y -395.061,Z 1282.845,A 0.000,B 0.000,C 90.000,E1 8.049} C_DIS
LIN {X -0.040,Y -395.056,Z 1282.845,A 0.000,B 0.000,C 90.000,E1 8.049} C_DIS
LIN {X -0.103,Y -395.158,Z 1282.844,A 0.000,B 0.000,C 90.000,E1 7.992} C_DIS
LIN {X -0.141,Y -395.188,Z 1282.844,A 0.000,B 0.000,C 90.000,E1 7.992} C_DIS
LIN {X -0.053,Y -396.324,Z 1282.843,A 0.000,B 0.000,C 90.000,E1 7.814} C_DIS
LIN {X 0.080,Y -399.331,Z 1282.842,A 0.000,B 0.000,C 90.000,E1 7.530} C_DIS
LIN {X -0.132,Y -405.257,Z 1282.840,A 0.000,B 0.000,C 90.000,E1 7.182} C_DIS
LIN {X -0.154,Y -410.590,Z 1282.838,A 0.000,B 0.000,C 90.000,E1 6.891} C_DIS
LIN {X -0.124,Y -416.843,Z 1282.836,A 0.000,B 0.000,C 90.000,E1 6.486} C_DIS
LIN {X -0.020,Y -424.654,Z 1282.833,A 0.000,B 0.000,C 90.000,E1 5.910} C_DIS
LIN {X 0.216,Y -432.460,Z 1282.829,A 0.000,B 0.000,C 90.000,E1 5.277} C_DIS
LIN {X -0.204,Y -441.853,Z 1282.825,A 0.000,B 0.000,C 90.000,E1 4.588} C_DIS
LIN {X 0.094,Y -450.897,Z 1282.821,A 0.000,B 0.000,C 90.000,E1 3.784} C_DIS
LIN {X 0.173,Y -455.390,Z 1282.819,A 0.000,B 0.000,C 90.000,E1 3.383} C_DIS
LIN {X 0.046,Y -461.196,Z 1282.816,A 0.000,B 0.000,C 90.000,E1 2.865} C_DIS
LIN {X 0.179,Y -466.865,Z 1282.813,A 0.000,B 0.000,C 90.000,E1 2.293} C_DIS
LIN {X -0.139,Y -473.686,Z 1282.809,A 0.000,B 0.000,C 90.000,E1 1.604} C_DIS
LIN {X 0.112,Y -479.035,Z 1282.806,A 0.000,B 0.000,C 90.000,E1 0.974} C_DIS
LIN {X -0.057,Y -485.199,Z 1282.801,A 0.000,B 0.000,C 90.000,E1 0.229} C_DIS
LIN {X 0.015,Y -490.734,Z 1282.797,A 0.000,B 0.000,C 90.000,E1 359.484} C_DIS
LIN {X 0.050,Y -496.892,Z 1282.792,A 0.000,B 0.000,C 90.000,E1 358.568} C_DIS
LIN {X -0.018,Y -501.691,Z 1282.788,A 0.000,B 0.000,C 90.000,E1 357.822} C_DIS
LIN {X 0.246,Y -505.317,Z 1282.785,A 0.000,B 0.000,C 90.000,E1 357.192} C_DIS
LIN {X -0.249,Y -509.556,Z 1282.781,A 0.000,B 0.000,C 90.000,E1 356.502} C_DIS
LIN {X -0.194,Y -513.505,Z 1282.776,A 0.000,B 0.000,C 90.000,E1 355.755} C_DIS
LIN {X -0.104,Y -517.166,Z 1282.772,A 0.000,B 0.000,C 90.000,E1 355.008} C_DIS
LIN {X -0.204,Y -519.950,Z 1282.769,A 0.000,B 0.000,C 90.000,E1 354.432} C_DIS
LIN {X -0.054,Y -523.193,Z 1282.765,A 0.000,B 0.000,C 90.000,E1 353.685} C_DIS
LIN {X 0.185,Y -526.204,Z 1282.761,A 0.000,B 0.000,C 90.000,E1 352.932} C_DIS
LIN {X 0.148,Y -528.462,Z 1282.758,A 0.000,B 0.000,C 90.000,E1 352.356} C_DIS
LIN {X 0.188,Y -532.606,Z 1282.751,A 0.000,B 0.000,C 90.000,E1 351.197} C_DIS
LIN {X 0.235,Y -535.325,Z 1282.746,A 0.000,B 0.000,C 90.000,E1 350.330} C_DIS
LIN {X -0.128,Y -537.837,Z 1282.742,A 0.000,B 0.000,C 90.000,E1 349.511} C_DIS
LIN {X 0.070,Y -540.053,Z 1282.737,A 0.000,B 0.000,C 90.000,E1 348.634} C_DIS
LIN {X -0.159,Y -542.723,Z 1282.731,A 0.000,B 0.000,C 90.000,E1 347.521} C_DIS
LIN {X 0.175,Y -545.102,Z 1282.724,A 0.000,B 0.000,C 90.000,E1 346.353} C_DIS
LIN {X -0.045,Y -546.131,Z 1282.721,A 0.000,B 0.000,C 90.000,E1 345.811} C_DIS
LIN {X -0.063,Y -547.953,Z 1282.715,A 0.000,B 0.000,C 90.000,E1 344.685} C_DIS
LIN {X -0.153,Y -549.034,Z 1282.710,A 0.000,B 0.000,C 90.000,E1 343.850} C_DIS
LIN {X 0.292,Y -549.882,Z 1282.706,A 0.000,B 0.000,C 90.000,E1 342.960} C_DIS
LIN {X -0.046,Y -550.785,Z 1282.699,A 0.000,B 0.000,C 90.000,E1 341.873} C_DIS
LIN {X -0.120,Y -551.117,Z 1282.695,A 0.000,B 0.000,C 90.000,E1 341.040} C_DIS
LIN {X -0.015,Y -551.085,Z 1282.690,A 0.000,B 0.000,C 90.000,E1 340.188} C_DIS
LIN {X -0.155,Y -550.545,Z 1282.684,A 0.000,B 0.000,C 90.000,E1 339.082} C_DIS
LIN {X -0.126,Y -550.105,Z 1282.681,A 0.000,B 0.000,C 90.000,E1 338.518} C_DIS
LIN {X -0.034,Y -549.073,Z 1282.676,A 0.000,B 0.000,C 90.000,E1 337.667} C_DIS
LIN {X -0.012,Y -548.281,Z 1282.673,A 0.000,B 0.000,C 90.000,E1 337.102} C_DIS
LIN {X 0.021,Y -546.265,Z 1282.667,A 0.000,B 0.000,C 90.000,E1 335.973} C_DIS
LIN {X 0.273,Y -544.599,Z 1282.662,A 0.000,B 0.000,C 90.000,E1 335.101} C_DIS
LIN {X -0.246,Y -541.498,Z 1282.656,A 0.000,B 0.000,C 90.000,E1 334.024} C_DIS
LIN {X 0.181,Y -539.024,Z 1282.651,A 0.000,B 0.000,C 90.000,E1 333.127} C_DIS
LIN {X -0.173,Y -535.011,Z 1282.645,A 0.000,B 0.000,C 90.000,E1 332.025} C_DIS
LIN {X 0.174,Y -531.660,Z 1282.640,A 0.000,B 0.000,C 90.000,E1 331.129} C_DIS
LIN {X 0.160,Y -528.453,Z 1282.636,A 0.000,B 0.000,C 90.000,E1 330.411} C_DIS
LIN {X 0.060,Y -523.286,Z 1282.630,A 0.000,B 0.000,C 90.000,E1 329.410} C_DIS
LIN {X -0.172,Y -515.955,Z 1282.623,A 0.000,B 0.000,C 90.000,E1 328.122} C_DIS
LIN {X -0.244,Y -511.023,Z 1282.618,A 0.000,B 0.000,C 90.000,E1 327.248} C_DIS
LIN {X 0.290,Y -505.230,Z 1282.611,A 0.000,B 0.000,C 90.000,E1 326.008} C_DIS
LIN {X 0.097,Y -504.580,Z 1282.611,A 0.000,B 0.000,C 90.000,E1 325.881} C_DIS
LIN {X 0.204,Y -502.143,Z 1282.607,A 0.000,B 0.000,C 90.000,E1 325.182} C_DIS
LIN {X -0.210,Y -499.959,Z 1282.601,A 0.000,B 0.000,C 90.000,E1 324.276} C_DIS
LIN {X 0.118,Y -498.568,Z 1282.596,A 0.000,B 0.000,C 90.000,E1 323.336} C_DIS
LIN {X 0.000,Y -497.621,Z 1282.590,A 0.000,B 0.000,C 90.000,E1 322.145} C_DIS
LIN {X -0.181,Y -497.183,Z 1282.580,A 0.000,B 0.000,C 90.000,E1 320.356} C_DIS
LIN {X -0.223,Y -497.383,Z 1282.571,A 0.000,B 0.000,C 90.000,E1 318.852} C_DIS
LIN {X -0.079,Y -497.648,Z 1282.561,A 0.000,B 0.000,C 90.000,E1 317.025} C_DIS
LIN {X 0.036,Y -497.915,Z 1282.551,A 0.000,B 0.000,C 90.000,E1 315.202} C_DIS
LIN {X 0.013,Y -498.232,Z 1282.539,A 0.000,B 0.000,C 90.000,E1 313.095} C_DIS
LIN {X -0.049,Y -498.581,Z 1282.531,A 0.000,B 0.000,C 90.000,E1 311.595} C_DIS
LIN {X -0.066,Y -498.844,Z 1282.523,A 0.000,B 0.000,C 90.000,E1 310.092} C_DIS
LIN {X -0.083,Y -499.037,Z 1282.514,A 0.000,B 0.000,C 90.000,E1 308.588} C_DIS
LIN {X -0.072,Y -498.985,Z 1282.509,A 0.000,B 0.000,C 90.000,E1 307.684} C_DIS
LIN {X -0.149,Y -498.554,Z 1282.504,A 0.000,B 0.000,C 90.000,E1 306.790} C_DIS
LIN {X -0.131,Y -497.698,Z 1282.499,A 0.000,B 0.000,C 90.000,E1 305.884} C_DIS
LIN {X 0.013,Y -496.770,Z 1282.496,A 0.000,B 0.000,C 90.000,E1 305.264} C_DIS
LIN {X 0.166,Y -496.108,Z 1282.494,A 0.000,B 0.000,C 90.000,E1 304.945} C_DIS
LIN {X 0.028,Y -495.204,Z 1282.493,A 0.000,B 0.000,C 90.000,E1 304.659} C_DIS
LIN {X -0.182,Y -494.587,Z 1282.492,A 0.000,B 0.000,C 90.000,E1 304.532} C_DIS
LIN {X 0.114,Y -478.349,Z 1282.476,A 0.000,B 0.000,C 90.000,E1 301.592} C_DIS
LIN {X 0.155,Y -463.944,Z 1282.459,A 0.000,B 0.000,C 90.000,E1 298.615} C_DIS
LIN {X 0.076,Y -451.338,Z 1282.442,A 0.000,B 0.000,C 90.000,E1 295.591} C_DIS
LIN {X 0.134,Y -439.917,Z 1282.424,A 0.000,B 0.000,C 90.000,E1 292.333} C_DIS
LIN {X 0.097,Y -430.288,Z 1282.406,A 0.000,B 0.000,C 90.000,E1 289.033} C_DIS
LIN {X -0.104,Y -421.674,Z 1282.385,A 0.000,B 0.000,C 90.000,E1 285.371} C_DIS
LIN {X -0.098,Y -414.052,Z 1282.361,A 0.000,B 0.000,C 90.000,E1 280.950} C_DIS
LIN {X -0.101,Y -408.337,Z 1282.330,A 0.000,B 0.000,C 90.000,E1 275.448} C_DIS
LIN {X -0.124,Y -410.503,Z 1282.257,A 0.000,B 0.000,C 90.000,E1 262.299} C_DIS
LIN {X 0.094,Y -416.930,Z 1282.230,A 0.000,B 0.000,C 90.000,E1 257.465} C_DIS
LIN {X 0.212,Y -424.954,Z 1282.208,A 0.000,B 0.000,C 90.000,E1 253.378} C_DIS
LIN {X 0.192,Y -434.437,Z 1282.187,A 0.000,B 0.000,C 90.000,E1 249.699} C_DIS
LIN {X -0.044,Y -444.907,Z 1282.169,A 0.000,B 0.000,C 90.000,E1 246.433} C_DIS
LIN {X 0.134,Y -456.560,Z 1282.152,A 0.000,B 0.000,C 90.000,E1 243.332} C_DIS
LIN {X -0.009,Y -461.278,Z 1282.146,A 0.000,B 0.000,C 90.000,E1 242.231} C_DIS
LIN {X 0.113,Y -462.196,Z 1282.144,A 0.000,B 0.000,C 90.000,E1 241.897} C_DIS
LIN {X 0.020,Y -462.780,Z 1282.142,A 0.000,B 0.000,C 90.000,E1 241.591} C_DIS
LIN {X -0.123,Y -463.508,Z 1282.139,A 0.000,B 0.000,C 90.000,E1 240.973} C_DIS
LIN {X 0.061,Y -464.006,Z 1282.133,A 0.000,B 0.000,C 90.000,E1 239.999} C_DIS
LIN {X -0.155,Y -464.014,Z 1282.128,A 0.000,B 0.000,C 90.000,E1 239.076} C_DIS
LIN {X 0.008,Y -463.474,Z 1282.121,A 0.000,B 0.000,C 90.000,E1 237.788} C_DIS
LIN {X 0.040,Y -462.354,Z 1282.110,A 0.000,B 0.000,C 90.000,E1 235.881} C_DIS
LIN {X 0.056,Y -460.905,Z 1282.096,A 0.000,B 0.000,C 90.000,E1 233.336} C_DIS
LIN {X -0.189,Y -460.006,Z 1282.086,A 0.000,B 0.000,C 90.000,E1 231.457} C_DIS
LIN {X 0.242,Y -459.061,Z 1282.072,A 0.000,B 0.000,C 90.000,E1 228.852} C_DIS
LIN {X -0.119,Y -458.377,Z 1282.059,A 0.000,B 0.000,C 90.000,E1 226.662} C_DIS
LIN {X -0.146,Y -457.880,Z 1282.045,A 0.000,B 0.000,C 90.000,E1 224.109} C_DIS
LIN {X 0.004,Y -458.353,Z 1282.024,A 0.000,B 0.000,C 90.000,E1 220.253} C_DIS
LIN {X -0.004,Y -458.940,Z 1282.013,A 0.000,B 0.000,C 90.000,E1 218.338} C_DIS
LIN {X 0.090,Y -463.782,Z 1281.978,A 0.000,B 0.000,C 90.000,E1 211.957} C_DIS
LIN {X -0.088,Y -466.100,Z 1281.967,A 0.000,B 0.000,C 90.000,E1 210.079} C_DIS
LIN {X 0.262,Y -469.057,Z 1281.953,A 0.000,B 0.000,C 90.000,E1 207.513} C_DIS
LIN {X 0.095,Y -471.998,Z 1281.941,A 0.000,B 0.000,C 90.000,E1 205.335} C_DIS
LIN {X 0.069,Y -474.819,Z 1281.930,A 0.000,B 0.000,C 90.000,E1 203.462} C_DIS
LIN {X 0.073,Y -478.686,Z 1281.917,A 0.000,B 0.000,C 90.000,E1 200.972} C_DIS
LIN {X 0.130,Y -483.294,Z 1281.901,A 0.000,B 0.000,C 90.000,E1 198.181} C_DIS
LIN {X -0.161,Y -486.022,Z 1281.893,A 0.000,B 0.000,C 90.000,E1 196.677} C_DIS
LIN {X -0.071,Y -488.785,Z 1281.884,A 0.000,B 0.000,C 90.000,E1 195.134} C_DIS
LIN {X -0.140,Y -492.607,Z 1281.872,A 0.000,B 0.000,C 90.000,E1 193.008} C_DIS
LIN {X -0.135,Y -495.974,Z 1281.862,A 0.000,B 0.000,C 90.000,E1 191.186} C_DIS
LIN {X -0.080,Y -498.737,Z 1281.854,A 0.000,B 0.000,C 90.000,E1 189.670} C_DIS
LIN {X -0.133,Y -502.169,Z 1281.844,A 0.000,B 0.000,C 90.000,E1 187.871} C_DIS
LIN {X -0.116,Y -504.968,Z 1281.835,A 0.000,B 0.000,C 90.000,E1 186.372} C_DIS
LIN {X -0.094,Y -507.622,Z 1281.827,A 0.000,B 0.000,C 90.000,E1 184.878} C_DIS
LIN {X -0.015,Y -510.313,Z 1281.819,A 0.000,B 0.000,C 90.000,E1 183.383} C_DIS
LIN {X 0.018,Y -513.329,Z 1281.809,A 0.000,B 0.000,C 90.000,E1 181.604} C_DIS
LIN {X 0.157,Y -515.685,Z 1281.801,A 0.000,B 0.000,C 90.000,E1 180.115} C_DIS
LIN {X -0.242,Y -518.358,Z 1281.791,A 0.000,B 0.000,C 90.000,E1 178.396} C_DIS
LIN {X 0.055,Y -520.000,Z 1281.784,A 0.000,B 0.000,C 90.000,E1 177.192} C_DIS
LIN {X -0.162,Y -521.720,Z 1281.776,A 0.000,B 0.000,C 90.000,E1 175.755} C_DIS
LIN {X 0.180,Y -522.882,Z 1281.770,A 0.000,B 0.000,C 90.000,E1 174.552} C_DIS
LIN {X 0.118,Y -523.735,Z 1281.763,A 0.000,B 0.000,C 90.000,E1 173.394} C_DIS
LIN {X 0.023,Y -524.583,Z 1281.755,A 0.000,B 0.000,C 90.000,E1 171.951} C_DIS
LIN {X -0.002,Y -524.920,Z 1281.749,A 0.000,B 0.000,C 90.000,E1 170.792} C_DIS
LIN {X -0.028,Y -525.025,Z 1281.742,A 0.000,B 0.000,C 90.000,E1 169.634} C_DIS
LIN {X 0.005,Y -525.032,Z 1281.739,A 0.000,B 0.000,C 90.000,E1 169.050} C_DIS
LIN {X 0.099,Y -524.436,Z 1281.729,A 0.000,B 0.000,C 90.000,E1 167.297} C_DIS
LIN {X -0.091,Y -523.330,Z 1281.720,A 0.000,B 0.000,C 90.000,E1 165.574} C_DIS
LIN {X 0.069,Y -522.537,Z 1281.713,A 0.000,B 0.000,C 90.000,E1 164.393} C_DIS
LIN {X -0.015,Y -521.096,Z 1281.702,A 0.000,B 0.000,C 90.000,E1 162.362} C_DIS
LIN {X 0.041,Y -520.180,Z 1281.692,A 0.000,B 0.000,C 90.000,E1 160.604} C_DIS
LIN {X -0.034,Y -520.230,Z 1281.686,A 0.000,B 0.000,C 90.000,E1 159.444} C_DIS
LIN {X 0.041,Y -521.208,Z 1281.678,A 0.000,B 0.000,C 90.000,E1 157.975} C_DIS
LIN {X -0.137,Y -522.088,Z 1281.674,A 0.000,B 0.000,C 90.000,E1 157.411} C_DIS
LIN {X 0.174,Y -523.221,Z 1281.671,A 0.000,B 0.000,C 90.000,E1 156.794} C_DIS
LIN {X 0.012,Y -524.702,Z 1281.668,A 0.000,B 0.000,C 90.000,E1 156.230} C_DIS
LIN {X -0.141,Y -526.638,Z 1281.665,A 0.000,B 0.000,C 90.000,E1 155.665} C_DIS
LIN {X 0.044,Y -529.762,Z 1281.661,A 0.000,B 0.000,C 90.000,E1 154.921} C_DIS
LIN {X 0.009,Y -533.692,Z 1281.657,A 0.000,B 0.000,C 90.000,E1 154.204} C_DIS
LIN {X 0.202,Y -535.407,Z 1281.655,A 0.000,B 0.000,C 90.000,E1 153.896} C_DIS
LIN {X -0.053,Y -542.702,Z 1281.650,A 0.000,B 0.000,C 90.000,E1 152.948} C_DIS
LIN {X 0.064,Y -549.896,Z 1281.645,A 0.000,B 0.000,C 90.000,E1 152.103} C_DIS
LIN {X -0.231,Y -566.344,Z 1281.636,A 0.000,B 0.000,C 90.000,E1 150.461} C_DIS
LIN {X 0.108,Y -576.665,Z 1281.630,A 0.000,B 0.000,C 90.000,E1 149.410} C_DIS
LIN {X -0.094,Y -584.322,Z 1281.626,A 0.000,B 0.000,C 90.000,E1 148.663} C_DIS
LIN {X -0.112,Y -592.942,Z 1281.621,A 0.000,B 0.000,C 90.000,E1 147.740} C_DIS
LIN {X 0.216,Y -599.970,Z 1281.616,A 0.000,B 0.000,C 90.000,E1 146.914} C_DIS
LIN {X -0.176,Y -605.343,Z 1281.613,A 0.000,B 0.000,C 90.000,E1 146.294} C_DIS
LIN {X 0.315,Y -610.222,Z 1281.609,A 0.000,B 0.000,C 90.000,E1 145.595} C_DIS
LIN {X 0.059,Y -613.003,Z 1281.607,A 0.000,B 0.000,C 90.000,E1 145.229} C_DIS
LIN {X -0.129,Y -617.264,Z 1281.603,A 0.000,B 0.000,C 90.000,E1 144.609} C_DIS
LIN {X 0.132,Y -620.497,Z 1281.600,A 0.000,B 0.000,C 90.000,E1 144.069} C_DIS
LIN {X 0.258,Y -624.270,Z 1281.597,A 0.000,B 0.000,C 90.000,E1 143.417} C_DIS
LIN {X -0.091,Y -628.461,Z 1281.593,A 0.000,B 0.000,C 90.000,E1 142.683} C_DIS
LIN {X -0.046,Y -633.974,Z 1281.586,A 0.000,B 0.000,C 90.000,E1 141.537} C_DIS
LIN {X 0.086,Y -637.768,Z 1281.581,A 0.000,B 0.000,C 90.000,E1 140.642} C_DIS
LIN {X -0.041,Y -639.814,Z 1281.579,A 0.000,B 0.000,C 90.000,E1 140.150} C_DIS
LIN {X 0.076,Y -643.628,Z 1281.573,A 0.000,B 0.000,C 90.000,E1 139.138} C_DIS
LIN {X -0.242,Y -648.088,Z 1281.566,A 0.000,B 0.000,C 90.000,E1 137.919} C_DIS
LIN {X -0.002,Y -651.419,Z 1281.561,A 0.000,B 0.000,C 90.000,E1 136.905} C_DIS
LIN {X 0.242,Y -655.540,Z 1281.554,A 0.000,B 0.000,C 90.000,E1 135.648} C_DIS
LIN {X 0.016,Y -662.146,Z 1281.543,A 0.000,B 0.000,C 90.000,E1 133.704} C_DIS
LIN {X -0.011,Y -666.309,Z 1281.536,A 0.000,B 0.000,C 90.000,E1 132.486} C_DIS
LIN {X -0.020,Y -669.625,Z 1281.531,A 0.000,B 0.000,C 90.000,E1 131.515} C_DIS
LIN {X -0.352,Y -674.276,Z 1281.523,A 0.000,B 0.000,C 90.000,E1 130.092} C_DIS
LIN {X 0.338,Y -678.002,Z 1281.516,A 0.000,B 0.000,C 90.000,E1 128.830} C_DIS
LIN {X 0.110,Y -680.800,Z 1281.511,A 0.000,B 0.000,C 90.000,E1 127.890} C_DIS
LIN {X -0.082,Y -683.474,Z 1281.505,A 0.000,B 0.000,C 90.000,E1 126.950} C_DIS
LIN {X -0.245,Y -685.972,Z 1281.500,A 0.000,B 0.000,C 90.000,E1 126.011} C_DIS
LIN {X -0.194,Y -688.890,Z 1281.493,A 0.000,B 0.000,C 90.000,E1 124.818} C_DIS
LIN {X -0.123,Y -691.026,Z 1281.488,A 0.000,B 0.000,C 90.000,E1 123.865} C_DIS
LIN {X -0.241,Y -692.486,Z 1281.484,A 0.000,B 0.000,C 90.000,E1 123.166} C_DIS
LIN {X 0.115,Y -694.713,Z 1281.478,A 0.000,B 0.000,C 90.000,E1 121.957} C_DIS
LIN {X -0.085,Y -696.698,Z 1281.471,A 0.000,B 0.000,C 90.000,E1 120.797} C_DIS
LIN {X -0.273,Y -698.167,Z 1281.466,A 0.000,B 0.000,C 90.000,E1 119.873} C_DIS
LIN {X -0.176,Y -699.778,Z 1281.459,A 0.000,B 0.000,C 90.000,E1 118.693} C_DIS
LIN {X 0.289,Y -700.794,Z 1281.454,A 0.000,B 0.000,C 90.000,E1 117.719} C_DIS
LIN {X -0.135,Y -701.366,Z 1281.450,A 0.000,B 0.000,C 90.000,E1 117.052} C_DIS
LIN {X 0.027,Y -701.547,Z 1281.445,A 0.000,B 0.000,C 90.000,E1 116.104} C_DIS
LIN {X 0.303,Y -701.571,Z 1281.444,A 0.000,B 0.000,C 90.000,E1 115.848} C_DIS
LIN {X 0.197,Y -701.218,Z 1281.440,A 0.000,B 0.000,C 90.000,E1 115.155} C_DIS
LIN {X -0.183,Y -700.774,Z 1281.437,A 0.000,B 0.000,C 90.000,E1 114.719} C_DIS
LIN {X -0.276,Y -700.051,Z 1281.435,A 0.000,B 0.000,C 90.000,E1 114.259} C_DIS
LIN {X -0.007,Y -699.398,Z 1281.433,A 0.000,B 0.000,C 90.000,E1 114.003} C_DIS
LIN {X 0.241,Y -697.607,Z 1281.431,A 0.000,B 0.000,C 90.000,E1 113.515} C_DIS
LIN {X 0.372,Y -696.909,Z 1281.430,A 0.000,B 0.000,C 90.000,E1 113.387} C_DIS
LIN {X -0.035,Y -693.352,Z 1281.427,A 0.000,B 0.000,C 90.000,E1 112.950} C_DIS
LIN {X 0.088,Y -692.165,Z 1281.427,A 0.000,B 0.000,C 90.000,E1 112.823} C_DIS
LIN {X -0.050,Y -690.338,Z 1281.426,A 0.000,B 0.000,C 90.000,E1 112.717} C_DIS
LIN {X 0.079,Y -687.725,Z 1281.426,A 0.000,B 0.000,C 90.000,E1 112.589} C_DIS
LIN {X -0.173,Y -683.432,Z 1281.424,A 0.000,B 0.000,C 90.000,E1 112.386} C_DIS
LIN {X 0.294,Y -679.150,Z 1281.424,A 0.000,B 0.000,C 90.000,E1 112.206} C_DIS
LIN {X -0.060,Y -677.623,Z 1281.423,A 0.000,B 0.000,C 90.000,E1 112.206} C_DIS
LIN {X 0.079,Y -670.906,Z 1281.423,A 0.000,B 0.000,C 90.000,E1 112.099} C_DIS
LIN {X 0.154,Y -668.122,Z 1281.423,A 0.000,B 0.000,C 90.000,E1 112.078} C_DIS
LIN {X 0.101,Y -664.272,Z 1281.423,A 0.000,B 0.000,C 90.000,E1 112.078} C_DIS
LIN {X 0.048,Y -639.533,Z 1281.423,A 0.000,B 0.000,C 90.000,E1 112.078} C_DIS
LIN {X -0.053,Y -638.807,Z 1281.423,A 0.000,B 0.000,C 90.000,E1 112.078} C_DIS
LIN {X 0.148,Y -636.403,Z 1281.422,A 0.000,B 0.000,C 90.000,E1 111.972} C_DIS
LIN {X 0.102,Y -636.318,Z 1281.422,A 0.000,B 0.000,C 90.000,E1 111.972} C_DIS
LIN {X -0.013,Y -636.883,Z 1281.421,A 0.000,B 0.000,C 90.000,E1 111.770} C_DIS
LIN {X 0.006,Y -637.490,Z 1281.420,A 0.000,B 0.000,C 90.000,E1 111.642} C_DIS
LIN {X -0.297,Y -642.795,Z 1281.416,A 0.000,B 0.000,C 90.000,E1 110.918} C_DIS
LIN {X 0.194,Y -646.452,Z 1281.413,A 0.000,B 0.000,C 90.000,E1 110.375} C_DIS
LIN {X 0.106,Y -649.842,Z 1281.411,A 0.000,B 0.000,C 90.000,E1 109.885} C_DIS
LIN {X 0.078,Y -653.474,Z 1281.407,A 0.000,B 0.000,C 90.000,E1 109.268} C_DIS
LIN {X 0.030,Y -656.112,Z 1281.404,A 0.000,B 0.000,C 90.000,E1 108.779} C_DIS
LIN {X -0.122,Y -659.642,Z 1281.400,A 0.000,B 0.000,C 90.000,E1 108.055} C_DIS
LIN {X -0.244,Y -662.893,Z 1281.396,A 0.000,B 0.000,C 90.000,E1 107.330} C_DIS
LIN {X 0.198,Y -664.892,Z 1281.394,A 0.000,B 0.000,C 90.000,E1 106.804} C_DIS
LIN {X 0.211,Y -666.672,Z 1281.391,A 0.000,B 0.000,C 90.000,E1 106.315} C_DIS
LIN {X -0.030,Y -668.964,Z 1281.387,A 0.000,B 0.000,C 90.000,E1 105.607} C_DIS
LIN {X -0.176,Y -670.322,Z 1281.384,A 0.000,B 0.000,C 90.000,E1 105.134} C_DIS
LIN {X -0.208,Y -671.932,Z 1281.380,A 0.000,B 0.000,C 90.000,E1 104.411} C_DIS
LIN {X 0.254,Y -673.081,Z 1281.376,A 0.000,B 0.000,C 90.000,E1 103.647} C_DIS
LIN {X 0.134,Y -673.668,Z 1281.373,A 0.000,B 0.000,C 90.000,E1 103.175} C_DIS
LIN {X 0.016,Y -674.039,Z 1281.371,A 0.000,B 0.000,C 90.000,E1 102.703} C_DIS
LIN {X -0.300,Y -674.248,Z 1281.367,A 0.000,B 0.000,C 90.000,E1 102.007} C_DIS
LIN {X 0.247,Y -674.190,Z 1281.364,A 0.000,B 0.000,C 90.000,E1 101.478} C_DIS
LIN {X -0.058,Y -673.639,Z 1281.360,A 0.000,B 0.000,C 90.000,E1 100.782} C_DIS
LIN {X -0.180,Y -673.075,Z 1281.357,A 0.000,B 0.000,C 90.000,E1 100.310} C_DIS
LIN {X 0.236,Y -672.221,Z 1281.355,A 0.000,B 0.000,C 90.000,E1 99.792} C_DIS
LIN {X 0.098,Y -671.175,Z 1281.352,A 0.000,B 0.000,C 90.000,E1 99.321} C_DIS
LIN {X -0.156,Y -669.795,Z 1281.349,A 0.000,B 0.000,C 90.000,E1 98.859} C_DIS
LIN {X 0.248,Y -668.059,Z 1281.347,A 0.000,B 0.000,C 90.000,E1 98.341} C_DIS
LIN {X 0.072,Y -666.031,Z 1281.344,A 0.000,B 0.000,C 90.000,E1 97.871} C_DIS
LIN {X -0.204,Y -664.299,Z 1281.342,A 0.000,B 0.000,C 90.000,E1 97.530} C_DIS
LIN {X 0.164,Y -661.726,Z 1281.339,A 0.000,B 0.000,C 90.000,E1 97.011} C_DIS
LIN {X -0.143,Y -658.821,Z 1281.336,A 0.000,B 0.000,C 90.000,E1 96.549} C_DIS
LIN {X 0.152,Y -654.654,Z 1281.333,A 0.000,B 0.000,C 90.000,E1 95.910} C_DIS
LIN {X -0.204,Y -650.998,Z 1281.330,A 0.000,B 0.000,C 90.000,E1 95.448} C_DIS
LIN {X 0.008,Y -647.042,Z 1281.328,A 0.000,B 0.000,C 90.000,E1 94.935} C_DIS
LIN {X 0.130,Y -641.469,Z 1281.324,A 0.000,B 0.000,C 90.000,E1 94.302} C_DIS
LIN {X 0.235,Y -635.358,Z 1281.321,A 0.000,B 0.000,C 90.000,E1 93.669} C_DIS
LIN {X 0.127,Y -630.570,Z 1281.318,A 0.000,B 0.000,C 90.000,E1 93.212} C_DIS
LIN {X -0.087,Y -623.972,Z 1281.315,A 0.000,B 0.000,C 90.000,E1 92.636} C_DIS
LIN {X 0.085,Y -615.821,Z 1281.311,A 0.000,B 0.000,C 90.000,E1 91.949} C_DIS
LIN {X -0.173,Y -608.523,Z 1281.308,A 0.000,B 0.000,C 90.000,E1 91.432} C_DIS
LIN {X 0.290,Y -602.253,Z 1281.306,A 0.000,B 0.000,C 90.000,E1 90.974} C_DIS
LIN {X 0.074,Y -596.196,Z 1281.304,A 0.000,B 0.000,C 90.000,E1 90.630} C_DIS
LIN {X 0.008,Y -589.334,Z 1281.302,A 0.000,B 0.000,C 90.000,E1 90.286} C_DIS
LIN {X -0.191,Y -581.947,Z 1281.300,A 0.000,B 0.000,C 90.000,E1 90.000} C_DIS
LIN {X 0.069,Y -576.669,Z 1281.299,A 0.000,B 0.000,C 90.000,E1 89.771} C_DIS
LIN {X -0.162,Y -571.648,Z 1281.297,A 0.000,B 0.000,C 90.000,E1 89.542} C_DIS
LIN {X 0.163,Y -570.736,Z 1281.297,A 0.000,B 0.000,C 90.000,E1 89.427} C_DIS
LIN {X 0.021,Y -569.422,Z 1281.296,A 0.000,B 0.000,C 90.000,E1 89.198} C_DIS
LIN {X -0.248,Y -569.056,Z 1281.293,A 0.000,B 0.000,C 90.000,E1 88.797} C_DIS
LIN {X 0.167,Y -571.996,Z 1281.273,A 0.000,B 0.000,C 90.000,E1 85.065} C_DIS
LIN {X 0.081,Y -574.040,Z 1281.262,A 0.000,B 0.000,C 90.000,E1 83.166} C_DIS
LIN {X 0.185,Y -576.273,Z 1281.252,A 0.000,B 0.000,C 90.000,E1 81.254} C_DIS
LIN {X -0.203,Y -577.491,Z 1281.245,A 0.000,B 0.000,C 90.000,E1 80.208} C_DIS
LIN {X -0.008,Y -578.604,Z 1281.240,A 0.000,B 0.000,C 90.000,E1 79.106} C_DIS
LIN {X -0.155,Y -580.256,Z 1281.229,A 0.000,B 0.000,C 90.000,E1 77.229} C_DIS
LIN {X 0.068,Y -581.604,Z 1281.220,A 0.000,B 0.000,C 90.000,E1 75.589} C_DIS
LIN {X -0.185,Y -582.552,Z 1281.213,A 0.000,B 0.000,C 90.000,E1 74.267} C_DIS
LIN {X -0.014,Y -583.382,Z 1281.205,A 0.000,B 0.000,C 90.000,E1 72.906} C_DIS
LIN {X 0.177,Y -584.478,Z 1281.196,A 0.000,B 0.000,C 90.000,E1 71.275} C_DIS
LIN {X -0.164,Y -585.306,Z 1281.187,A 0.000,B 0.000,C 90.000,E1 69.699} C_DIS
LIN {X -0.120,Y -586.688,Z 1281.174,A 0.000,B 0.000,C 90.000,E1 67.283} C_DIS
LIN {X -0.102,Y -588.113,Z 1281.163,A 0.000,B 0.000,C 90.000,E1 65.409} C_DIS
LIN {X 0.298,Y -589.352,Z 1281.154,A 0.000,B 0.000,C 90.000,E1 63.768} C_DIS
LIN {X 0.350,Y -590.940,Z 1281.144,A 0.000,B 0.000,C 90.000,E1 61.897} C_DIS
LIN {X 0.016,Y -592.497,Z 1281.135,A 0.000,B 0.000,C 90.000,E1 60.333} C_DIS
LIN {X 0.107,Y -594.683,Z 1281.123,A 0.000,B 0.000,C 90.000,E1 58.201} C_DIS
LIN {X -0.158,Y -596.619,Z 1281.113,A 0.000,B 0.000,C 90.000,E1 56.373} C_DIS
LIN {X -0.184,Y -597.941,Z 1281.106,A 0.000,B 0.000,C 90.000,E1 55.055} C_DIS
LIN {X 0.162,Y -599.146,Z 1281.099,A 0.000,B 0.000,C 90.000,E1 53.703} C_DIS
LIN {X 0.046,Y -599.855,Z 1281.094,A 0.000,B 0.000,C 90.000,E1 52.924} C_DIS
LIN {X -0.031,Y -601.349,Z 1281.084,A 0.000,B 0.000,C 90.000,E1 51.090} C_DIS
LIN {X 0.031,Y -601.978,Z 1281.078,A 0.000,B 0.000,C 90.000,E1 50.033} C_DIS
LIN {X -0.079,Y -602.332,Z 1281.074,A 0.000,B 0.000,C 90.000,E1 49.256} C_DIS
LIN {X 0.184,Y -602.956,Z 1281.066,A 0.000,B 0.000,C 90.000,E1 47.919} C_DIS
LIN {X -0.182,Y -603.333,Z 1281.061,A 0.000,B 0.000,C 90.000,E1 46.905} C_DIS
LIN {X 0.108,Y -603.573,Z 1281.053,A 0.000,B 0.000,C 90.000,E1 45.567} C_DIS
LIN {X -0.034,Y -603.540,Z 1281.046,A 0.000,B 0.000,C 90.000,E1 44.271} C_DIS
LIN {X 0.259,Y -603.238,Z 1281.039,A 0.000,B 0.000,C 90.000,E1 42.933} C_DIS
LIN {X -0.107,Y -602.957,Z 1281.033,A 0.000,B 0.000,C 90.000,E1 41.919} C_DIS
LIN {X -0.272,Y -602.649,Z 1281.029,A 0.000,B 0.000,C 90.000,E1 41.148} C_DIS
LIN {X 0.053,Y -602.055,Z 1281.021,A 0.000,B 0.000,C 90.000,E1 39.806} C_DIS
LIN {X 0.368,Y -601.317,Z 1281.014,A 0.000,B 0.000,C 90.000,E1 38.463} C_DIS
LIN {X 0.042,Y -600.421,Z 1281.008,A 0.000,B 0.000,C 90.000,E1 37.443} C_DIS
LIN {X -0.061,Y -599.589,Z 1281.004,A 0.000,B 0.000,C 90.000,E1 36.664} C_DIS
LIN {X 0.071,Y -598.244,Z 1280.998,A 0.000,B 0.000,C 90.000,E1 35.598} C_DIS
LIN {X -0.054,Y -597.057,Z 1280.993,A 0.000,B 0.000,C 90.000,E1 34.818} C_DIS
LIN {X -0.302,Y -595.138,Z 1280.988,A 0.000,B 0.000,C 90.000,E1 33.785} C_DIS
LIN {X 0.031,Y -593.595,Z 1280.983,A 0.000,B 0.000,C 90.000,E1 32.959} C_DIS
LIN {X 0.137,Y -592.382,Z 1280.980,A 0.000,B 0.000,C 90.000,E1 32.418} C_DIS
LIN {X -0.296,Y -588.674,Z 1280.973,A 0.000,B 0.000,C 90.000,E1 31.131} C_DIS
LIN {X -0.345,Y -586.002,Z 1280.968,A 0.000,B 0.000,C 90.000,E1 30.335} C_DIS
LIN {X 0.213,Y -584.042,Z 1280.965,A 0.000,B 0.000,C 90.000,E1 29.745} C_DIS
LIN {X 0.247,Y -581.898,Z 1280.962,A 0.000,B 0.000,C 90.000,E1 29.205} C_DIS
LIN {X -0.085,Y -578.850,Z 1280.959,A 0.000,B 0.000,C 90.000,E1 28.565} C_DIS
LIN {X 0.189,Y -574.095,Z 1280.953,A 0.000,B 0.000,C 90.000,E1 27.590} C_DIS
LIN {X -0.029,Y -569.422,Z 1280.949,A 0.000,B 0.000,C 90.000,E1 26.796} C_DIS
LIN {X 0.221,Y -566.980,Z 1280.947,A 0.000,B 0.000,C 90.000,E1 26.360} C_DIS
LIN {X -0.139,Y -563.482,Z 1280.944,A 0.000,B 0.000,C 90.000,E1 25.848} C_DIS
LIN {X -0.112,Y -558.780,Z 1280.940,A 0.000,B 0.000,C 90.000,E1 25.155} C_DIS
LIN {X 0.086,Y -555.801,Z 1280.937,A 0.000,B 0.000,C 90.000,E1 24.719} C_DIS
LIN {X 0.158,Y -551.547,Z 1280.934,A 0.000,B 0.000,C 90.000,E1 24.155} C_DIS
LIN {X -0.302,Y -547.003,Z 1280.931,A 0.000,B 0.000,C 90.000,E1 23.643} C_DIS
LIN {X 0.131,Y -539.973,Z 1280.927,A 0.000,B 0.000,C 90.000,E1 22.770} C_DIS
LIN {X 0.089,Y -531.053,Z 1280.921,A 0.000,B 0.000,C 90.000,E1 21.791} C_DIS
LIN {X 0.005,Y -524.483,Z 1280.917,A 0.000,B 0.000,C 90.000,E1 21.099} C_DIS
LIN {X 0.043,Y -515.192,Z 1280.912,A 0.000,B 0.000,C 90.000,E1 20.120} C_DIS
LIN {X -0.088,Y -504.092,Z 1280.906,A 0.000,B 0.000,C 90.000,E1 19.033} C_DIS
LIN {X -0.016,Y -492.928,Z 1280.900,A 0.000,B 0.000,C 90.000,E1 17.946} C_DIS
LIN {X 0.000,Y -487.242,Z 1280.897,A 0.000,B 0.000,C 90.000,E1 17.402} C_DIS
LIN {X 0.029,Y -479.884,Z 1280.893,A 0.000,B 0.000,C 90.000,E1 16.732} C_DIS
LIN {X -0.060,Y -466.523,Z 1280.886,A 0.000,B 0.000,C 90.000,E1 15.552} C_DIS
LIN {X -0.015,Y -448.851,Z 1280.877,A 0.000,B 0.000,C 90.000,E1 13.939} C_DIS
LIN {X -0.117,Y -425.576,Z 1280.865,A 0.000,B 0.000,C 90.000,E1 11.658} C_DIS
LIN {X -0.045,Y -409.800,Z 1280.855,A 0.000,B 0.000,C 90.000,E1 9.962} C_DIS
LIN {X -0.132,Y -399.942,Z 1280.849,A 0.000,B 0.000,C 90.000,E1 8.859} C_DIS
LIN {X -0.173,Y -395.737,Z 1280.846,A 0.000,B 0.000,C 90.000,E1 8.276} C_DIS
LIN {X 0.102,Y -394.966,Z 1280.845,A 0.000,B 0.000,C 90.000,E1 8.049} C_DIS
LIN {X 0.065,Y -394.968,Z 1280.845,A 0.000,B 0.000,C 90.000,E1 8.049} C_DIS
LIN {X -0.087,Y -395.001,Z 1280.845,A 0.000,B 0.000,C 90.000,E1 8.049} C_DIS
LIN {X -0.126,Y -395.018,Z 1280.845,A 0.000,B 0.000,C 90.000,E1 8.049} C_DIS
LIN {X 0.115,Y -395.879,Z 1280.844,A 0.000,B 0.000,C 90.000,E1 7.871} C_DIS
LIN {X -0.103,Y -396.596,Z 1280.843,A 0.000,B 0.000,C 90.000,E1 7.814} C_DIS
LIN {X 0.062,Y -398.873,Z 1280.842,A 0.000,B 0.000,C 90.000,E1 7.587} C_DIS
LIN {X 0.095,Y -400.276,Z 1280.842,A 0.000,B 0.000,C 90.000,E1 7.473} C_DIS
LIN {X -0.097,Y -412.491,Z 1280.838,A 0.000,B 0.000,C 90.000,E1 6.777} C_DIS
LIN {X 0.182,Y -417.282,Z 1280.836,A 0.000,B 0.000,C 90.000,E1 6.429} C_DIS
LIN {X 0.193,Y -425.191,Z 1280.833,A 0.000,B 0.000,C 90.000,E1 5.853} C_DIS
LIN {X -0.091,Y -433.144,Z 1280.829,A 0.000,B 0.000,C 90.000,E1 5.277} C_DIS
LIN {X -0.097,Y -442.511,Z 1280.825,A 0.000,B 0.000,C 90.000,E1 4.531} C_DIS
LIN {X 0.183,Y -453.020,Z 1280.820,A 0.000,B 0.000,C 90.000,E1 3.612} C_DIS
LIN {X -0.042,Y -460.393,Z 1280.817,A 0.000,B 0.000,C 90.000,E1 2.980} C_DIS
LIN {X -0.146,Y -467.485,Z 1280.813,A 0.000,B 0.000,C 90.000,E1 2.293} C_DIS
LIN {X 0.205,Y -474.135,Z 1280.809,A 0.000,B 0.000,C 90.000,E1 1.547} C_DIS
LIN {X 0.034,Y -479.442,Z 1280.806,A 0.000,B 0.000,C 90.000,E1 0.974} C_DIS
LIN {X 0.016,Y -485.507,Z 1280.801,A 0.000,B 0.000,C 90.000,E1 0.229} C_DIS
LIN {X 0.017,Y -491.142,Z 1280.797,A 0.000,B 0.000,C 90.000,E1 359.484} C_DIS
LIN {X 0.056,Y -497.333,Z 1280.792,A 0.000,B 0.000,C 90.000,E1 358.568} C_DIS
LIN {X -0.009,Y -502.132,Z 1280.788,A 0.000,B 0.000,C 90.000,E1 357.822} C_DIS
LIN {X -0.246,Y -505.759,Z 1280.785,A 0.000,B 0.000,C 90.000,E1 357.249} C_DIS
LIN {X -0.231,Y -510.031,Z 1280.781,A 0.000,B 0.000,C 90.000,E1 356.502} C_DIS
LIN {X -0.172,Y -513.979,Z 1280.776,A 0.000,B 0.000,C 90.000,E1 355.755} C_DIS
LIN {X 0.220,Y -516.971,Z 1280.773,A 0.000,B 0.000,C 90.000,E1 355.122} C_DIS
LIN {X -0.172,Y -520.424,Z 1280.769,A 0.000,B 0.000,C 90.000,E1 354.432} C_DIS
LIN {X 0.272,Y -523.116,Z 1280.766,A 0.000,B 0.000,C 90.000,E1 353.799} C_DIS
LIN {X 0.216,Y -525.595,Z 1280.763,A 0.000,B 0.000,C 90.000,E1 353.223} C_DIS
LIN {X 0.173,Y -527.903,Z 1280.759,A 0.000,B 0.000,C 90.000,E1 352.648} C_DIS
LIN {X 0.201,Y -532.135,Z 1280.753,A 0.000,B 0.000,C 90.000,E1 351.489} C_DIS
LIN {X -0.285,Y -534.997,Z 1280.748,A 0.000,B 0.000,C 90.000,E1 350.679} C_DIS
LIN {X -0.126,Y -537.555,Z 1280.743,A 0.000,B 0.000,C 90.000,E1 349.803} C_DIS
LIN {X 0.067,Y -539.906,Z 1280.739,A 0.000,B 0.000,C 90.000,E1 348.926} C_DIS
LIN {X -0.081,Y -543.283,Z 1280.731,A 0.000,B 0.000,C 90.000,E1 347.521} C_DIS
LIN {X -0.269,Y -545.689,Z 1280.724,A 0.000,B 0.000,C 90.000,E1 346.408} C_DIS
LIN {X -0.089,Y -546.715,Z 1280.721,A 0.000,B 0.000,C 90.000,E1 345.825} C_DIS
LIN {X -0.108,Y -548.535,Z 1280.715,A 0.000,B 0.000,C 90.000,E1 344.700} C_DIS
LIN {X -0.201,Y -549.651,Z 1280.710,A 0.000,B 0.000,C 90.000,E1 343.866} C_DIS
LIN {X -0.123,Y -550.577,Z 1280.706,A 0.000,B 0.000,C 90.000,E1 343.015} C_DIS
LIN {X 0.076,Y -551.487,Z 1280.699,A 0.000,B 0.000,C 90.000,E1 341.873} C_DIS
LIN {X -0.083,Y -551.778,Z 1280.696,A 0.000,B 0.000,C 90.000,E1 341.329} C_DIS
LIN {X 0.282,Y -551.917,Z 1280.693,A 0.000,B 0.000,C 90.000,E1 340.732} C_DIS
LIN {X -0.122,Y -551.776,Z 1280.688,A 0.000,B 0.000,C 90.000,E1 339.934} C_DIS
LIN {X -0.007,Y -551.329,Z 1280.684,A 0.000,B 0.000,C 90.000,E1 339.082} C_DIS
LIN {X 0.098,Y -550.675,Z 1280.679,A 0.000,B 0.000,C 90.000,E1 338.230} C_DIS
LIN {X 0.157,Y -549.170,Z 1280.673,A 0.000,B 0.000,C 90.000,E1 337.102} C_DIS
LIN {X -0.058,Y -547.720,Z 1280.668,A 0.000,B 0.000,C 90.000,E1 336.282} C_DIS
LIN {X 0.215,Y -546.106,Z 1280.664,A 0.000,B 0.000,C 90.000,E1 335.409} C_DIS
LIN {X 0.218,Y -544.912,Z 1280.660,A 0.000,B 0.000,C 90.000,E1 334.845} C_DIS
LIN {X 0.211,Y -543.310,Z 1280.657,A 0.000,B 0.000,C 90.000,E1 334.280} C_DIS
LIN {X -0.042,Y -542.586,Z 1280.656,A 0.000,B 0.000,C 90.000,E1 334.024} C_DIS
LIN {X -0.086,Y -540.141,Z 1280.651,A 0.000,B 0.000,C 90.000,E1 333.179} C_DIS
LIN {X 0.056,Y -536.140,Z 1280.645,A 0.000,B 0.000,C 90.000,E1 332.025} C_DIS
LIN {X -0.195,Y -532.172,Z 1280.639,A 0.000,B 0.000,C 90.000,E1 331.051} C_DIS
LIN {X -0.202,Y -528.882,Z 1280.635,A 0.000,B 0.000,C 90.000,E1 330.333} C_DIS
LIN {X 0.021,Y -525.176,Z 1280.631,A 0.000,B 0.000,C 90.000,E1 329.587} C_DIS
LIN {X 0.099,Y -516.946,Z 1280.623,A 0.000,B 0.000,C 90.000,E1 328.122} C_DIS
LIN {X -0.028,Y -511.179,Z 1280.617,A 0.000,B 0.000,C 90.000,E1 327.120} C_DIS
LIN {X 0.029,Y -506.112,Z 1280.612,A 0.000,B 0.000,C 90.000,E1 326.087} C_DIS
LIN {X -0.267,Y -504.311,Z 1280.609,A 0.000,B 0.000,C 90.000,E1 325.674} C_DIS
LIN {X 0.129,Y -502.648,Z 1280.607,A 0.000,B 0.000,C 90.000,E1 325.182} C_DIS
LIN {X -0.279,Y -500.397,Z 1280.601,A 0.000,B 0.000,C 90.000,E1 324.276} C_DIS
LIN {X 0.056,Y -498.968,Z 1280.596,A 0.000,B 0.000,C 90.000,E1 323.336} C_DIS
LIN {X 0.248,Y -498.030,Z 1280.590,A 0.000,B 0.000,C 90.000,E1 322.110} C_DIS
LIN {X -0.228,Y -497.624,Z 1280.580,A 0.000,B 0.000,C 90.000,E1 320.356} C_DIS
LIN {X -0.126,Y -497.769,Z 1280.573,A 0.000,B 0.000,C 90.000,E1 319.138} C_DIS
LIN {X 0.035,Y -498.024,Z 1280.563,A 0.000,B 0.000,C 90.000,E1 317.310} C_DIS
LIN {X 0.169,Y -498.298,Z 1280.553,A 0.000,B 0.000,C 90.000,E1 315.486} C_DIS
LIN {X -0.049,Y -498.610,Z 1280.543,A 0.000,B 0.000,C 90.000,E1 313.704} C_DIS
LIN {X -0.244,Y -498.979,Z 1280.533,A 0.000,B 0.000,C 90.000,E1 311.919} C_DIS
LIN {X 0.074,Y -499.283,Z 1280.524,A 0.000,B 0.000,C 90.000,E1 310.378} C_DIS
LIN {X -0.065,Y -499.514,Z 1280.514,A 0.000,B 0.000,C 90.000,E1 308.588} C_DIS
LIN {X 0.131,Y -499.651,Z 1280.508,A 0.000,B 0.000,C 90.000,E1 307.363} C_DIS
LIN {X 0.159,Y -499.530,Z 1280.503,A 0.000,B 0.000,C 90.000,E1 306.457} C_DIS
LIN {X -0.214,Y -499.123,Z 1280.498,A 0.000,B 0.000,C 90.000,E1 305.598} C_DIS
LIN {X -0.058,Y -498.631,Z 1280.494,A 0.000,B 0.000,C 90.000,E1 304.978} C_DIS
LIN {X -0.315,Y -497.881,Z 1280.491,A 0.000,B 0.000,C 90.000,E1 304.405} C_DIS
LIN {X -0.034,Y -497.381,Z 1280.489,A 0.000,B 0.000,C 90.000,E1 304.072} C_DIS
LIN {X -0.167,Y -496.743,Z 1280.488,A 0.000,B 0.000,C 90.000,E1 303.785} C_DIS
LIN {X 0.111,Y -495.880,Z 1280.486,A 0.000,B 0.000,C 90.000,E1 303.452} C_DIS
LIN {X 0.178,Y -495.325,Z 1280.485,A 0.000,B 0.000,C 90.000,E1 303.293} C_DIS
LIN {X 0.036,Y -493.745,Z 1280.483,A 0.000,B 0.000,C 90.000,E1 303.007} C_DIS
LIN {X -0.206,Y -478.360,Z 1280.467,A 0.000,B 0.000,C 90.000,E1 300.129} C_DIS
LIN {X 0.039,Y -464.809,Z 1280.451,A 0.000,B 0.000,C 90.000,E1 297.129} C_DIS
LIN {X 0.221,Y -453.000,Z 1280.434,A 0.000,B 0.000,C 90.000,E1 294.079} C_DIS
LIN {X 0.014,Y -442.358,Z 1280.416,A 0.000,B 0.000,C 90.000,E1 290.865} C_DIS
LIN {X 0.177,Y -432.662,Z 1280.396,A 0.000,B 0.000,C 90.000,E1 287.221} C_DIS
LIN {X -0.071,Y -424.383,Z 1280.374,A 0.000,B 0.000,C 90.000,E1 283.244} C_DIS
LIN {X -0.100,Y -417.634,Z 1280.347,A 0.000,B 0.000,C 90.000,E1 278.511} C_DIS
LIN {X 0.010,Y -413.187,Z 1280.307,A 0.000,B 0.000,C 90.000,E1 271.318} C_DIS
LIN {X -0.037,Y -416.632,Z 1280.260,A 0.000,B 0.000,C 90.000,E1 262.761} C_DIS
LIN {X 0.039,Y -422.767,Z 1280.233,A 0.000,B 0.000,C 90.000,E1 257.993} C_DIS
LIN {X -0.089,Y -430.514,Z 1280.211,A 0.000,B 0.000,C 90.000,E1 253.976} C_DIS
LIN {X -0.016,Y -439.716,Z 1280.191,A 0.000,B 0.000,C 90.000,E1 250.315} C_DIS
LIN {X -0.051,Y -449.904,Z 1280.172,A 0.000,B 0.000,C 90.000,E1 247.050} C_DIS
LIN {X 0.069,Y -461.910,Z 1280.155,A 0.000,B 0.000,C 90.000,E1 243.819} C_DIS
LIN {X -0.015,Y -463.111,Z 1280.153,A 0.000,B 0.000,C 90.000,E1 243.512} C_DIS
LIN {X -0.097,Y -463.846,Z 1280.151,A 0.000,B 0.000,C 90.000,E1 243.204} C_DIS
LIN {X 0.033,Y -464.340,Z 1280.149,A 0.000,B 0.000,C 90.000,E1 242.871} C_DIS
LIN {X 0.088,Y -464.913,Z 1280.146,A 0.000,B 0.000,C 90.000,E1 242.231} C_DIS
LIN {X -0.119,Y -465.285,Z 1280.141,A 0.000,B 0.000,C 90.000,E1 241.307} C_DIS
LIN {X 0.087,Y -465.311,Z 1280.135,A 0.000,B 0.000,C 90.000,E1 240.333} C_DIS
LIN {X -0.115,Y -465.024,Z 1280.130,A 0.000,B 0.000,C 90.000,E1 239.410} C_DIS
LIN {X 0.063,Y -464.254,Z 1280.123,A 0.000,B 0.000,C 90.000,E1 238.122} C_DIS
LIN {X 0.232,Y -463.467,Z 1280.116,A 0.000,B 0.000,C 90.000,E1 236.834} C_DIS
LIN {X 0.129,Y -462.519,Z 1280.107,A 0.000,B 0.000,C 90.000,E1 235.261} C_DIS
LIN {X -0.224,Y -461.129,Z 1280.093,A 0.000,B 0.000,C 90.000,E1 232.763} C_DIS
LIN {X 0.180,Y -460.258,Z 1280.082,A 0.000,B 0.000,C 90.000,E1 230.803} C_DIS
LIN {X -0.152,Y -459.577,Z 1280.072,A 0.000,B 0.000,C 90.000,E1 228.933} C_DIS
LIN {X 0.109,Y -458.992,Z 1280.061,A 0.000,B 0.000,C 90.000,E1 226.986} C_DIS
LIN {X 0.101,Y -458.443,Z 1280.047,A 0.000,B 0.000,C 90.000,E1 224.433} C_DIS
LIN {X -0.040,Y -458.759,Z 1280.024,A 0.000,B 0.000,C 90.000,E1 220.297} C_DIS
LIN {X -0.049,Y -459.276,Z 1280.013,A 0.000,B 0.000,C 90.000,E1 218.382} C_DIS
LIN {X 0.040,Y -464.041,Z 1279.978,A 0.000,B 0.000,C 90.000,E1 212.005} C_DIS
LIN {X -0.142,Y -466.355,Z 1279.967,A 0.000,B 0.000,C 90.000,E1 210.129} C_DIS
LIN {X 0.052,Y -468.905,Z 1279.955,A 0.000,B 0.000,C 90.000,E1 207.897} C_DIS
LIN {X -0.121,Y -471.782,Z 1279.943,A 0.000,B 0.000,C 90.000,E1 205.720} C_DIS
LIN {X 0.008,Y -474.985,Z 1279.931,A 0.000,B 0.000,C 90.000,E1 203.515} C_DIS
LIN {X -0.162,Y -478.902,Z 1279.917,A 0.000,B 0.000,C 90.000,E1 201.046} C_DIS
LIN {X 0.066,Y -483.560,Z 1279.901,A 0.000,B 0.000,C 90.000,E1 198.236} C_DIS
LIN {X 0.108,Y -486.853,Z 1279.891,A 0.000,B 0.000,C 90.000,E1 196.386} C_DIS
LIN {X -0.133,Y -489.105,Z 1279.884,A 0.000,B 0.000,C 90.000,E1 195.190} C_DIS
LIN {X 0.183,Y -493.577,Z 1279.871,A 0.000,B 0.000,C 90.000,E1 192.715} C_DIS
LIN {X 0.212,Y -497.000,Z 1279.861,A 0.000,B 0.000,C 90.000,E1 190.894} C_DIS
LIN {X 0.129,Y -500.366,Z 1279.851,A 0.000,B 0.000,C 90.000,E1 189.095} C_DIS
LIN {X 0.120,Y -503.892,Z 1279.841,A 0.000,B 0.000,C 90.000,E1 187.296} C_DIS
LIN {X -0.266,Y -506.142,Z 1279.834,A 0.000,B 0.000,C 90.000,E1 186.144} C_DIS
LIN {X -0.174,Y -508.848,Z 1279.826,A 0.000,B 0.000,C 90.000,E1 184.645} C_DIS
LIN {X -0.110,Y -511.593,Z 1279.818,A 0.000,B 0.000,C 90.000,E1 183.154} C_DIS
LIN {X 0.031,Y -514.174,Z 1279.809,A 0.000,B 0.000,C 90.000,E1 181.661} C_DIS
LIN {X 0.117,Y -517.080,Z 1279.799,A 0.000,B 0.000,C 90.000,E1 179.885} C_DIS
LIN {X -0.194,Y -519.380,Z 1279.791,A 0.000,B 0.000,C 90.000,E1 178.453} C_DIS
LIN {X 0.119,Y -521.086,Z 1279.785,A 0.000,B 0.000,C 90.000,E1 177.249} C_DIS
LIN {X -0.078,Y -522.900,Z 1279.777,A 0.000,B 0.000,C 90.000,E1 175.812} C_DIS
LIN {X -0.237,Y -524.129,Z 1279.770,A 0.000,B 0.000,C 90.000,E1 174.666} C_DIS
LIN {X 0.235,Y -524.892,Z 1279.765,A 0.000,B 0.000,C 90.000,E1 173.742} C_DIS
LIN {X 0.200,Y -525.511,Z 1279.761,A 0.000,B 0.000,C 90.000,E1 172.875} C_DIS
LIN {X 0.115,Y -526.283,Z 1279.754,A 0.000,B 0.000,C 90.000,E1 171.724} C_DIS
LIN {X 0.108,Y -526.671,Z 1279.748,A 0.000,B 0.000,C 90.000,E1 170.566} C_DIS
LIN {X 0.220,Y -526.860,Z 1279.740,A 0.000,B 0.000,C 90.000,E1 169.106} C_DIS
LIN {X -0.176,Y -526.600,Z 1279.732,A 0.000,B 0.000,C 90.000,E1 167.701} C_DIS
LIN {X 0.032,Y -526.168,Z 1279.725,A 0.000,B 0.000,C 90.000,E1 166.520} C_DIS
LIN {X 0.253,Y -525.373,Z 1279.717,A 0.000,B 0.000,C 90.000,E1 165.046} C_DIS
LIN {X -0.067,Y -524.805,Z 1279.711,A 0.000,B 0.000,C 90.000,E1 163.921} C_DIS
LIN {X 0.057,Y -523.729,Z 1279.698,A 0.000,B 0.000,C 90.000,E1 161.583} C_DIS
LIN {X -0.131,Y -523.588,Z 1279.693,A 0.000,B 0.000,C 90.000,E1 160.732} C_DIS
LIN {X 0.167,Y -524.305,Z 1279.683,A 0.000,B 0.000,C 90.000,E1 158.954} C_DIS
LIN {X -0.183,Y -524.850,Z 1279.680,A 0.000,B 0.000,C 90.000,E1 158.411} C_DIS
LIN {X 0.149,Y -525.807,Z 1279.677,A 0.000,B 0.000,C 90.000,E1 157.794} C_DIS
LIN {X 0.175,Y -527.534,Z 1279.672,A 0.000,B 0.000,C 90.000,E1 156.922} C_DIS
LIN {X 0.222,Y -530.220,Z 1279.667,A 0.000,B 0.000,C 90.000,E1 156.049} C_DIS
LIN {X -0.230,Y -531.808,Z 1279.665,A 0.000,B 0.000,C 90.000,E1 155.665} C_DIS
LIN {X 0.153,Y -534.386,Z 1279.661,A 0.000,B 0.000,C 90.000,E1 155.049} C_DIS
LIN {X -0.278,Y -536.504,Z 1279.659,A 0.000,B 0.000,C 90.000,E1 154.665} C_DIS
LIN {X -0.114,Y -539.932,Z 1279.656,A 0.000,B 0.000,C 90.000,E1 154.076} C_DIS
LIN {X 0.151,Y -545.990,Z 1279.651,A 0.000,B 0.000,C 90.000,E1 153.204} C_DIS
LIN {X 0.276,Y -551.837,Z 1279.647,A 0.000,B 0.000,C 90.000,E1 152.487} C_DIS
LIN {X 0.279,Y -569.525,Z 1279.637,A 0.000,B 0.000,C 90.000,E1 150.589} C_DIS
LIN {X 0.056,Y -577.223,Z 1279.632,A 0.000,B 0.000,C 90.000,E1 149.822} C_DIS
LIN {X 0.060,Y -585.734,Z 1279.627,A 0.000,B 0.000,C 90.000,E1 148.918} C_DIS
LIN {X -0.021,Y -590.433,Z 1279.625,A 0.000,B 0.000,C 90.000,E1 148.408} C_DIS
LIN {X -0.173,Y -596.124,Z 1279.621,A 0.000,B 0.000,C 90.000,E1 147.788} C_DIS
LIN {X -0.100,Y -601.794,Z 1279.617,A 0.000,B 0.000,C 90.000,E1 147.120} C_DIS
LIN {X 0.356,Y -606.905,Z 1279.614,A 0.000,B 0.000,C 90.000,E1 146.421} C_DIS
LIN {X 0.015,Y -611.638,Z 1279.610,A 0.000,B 0.000,C 90.000,E1 145.801} C_DIS
LIN {X 0.272,Y -614.249,Z 1279.608,A 0.000,B 0.000,C 90.000,E1 145.388} C_DIS
LIN {X 0.011,Y -617.593,Z 1279.605,A 0.000,B 0.000,C 90.000,E1 144.895} C_DIS
LIN {X 0.093,Y -622.249,Z 1279.601,A 0.000,B 0.000,C 90.000,E1 144.116} C_DIS
LIN {X -0.133,Y -625.826,Z 1279.597,A 0.000,B 0.000,C 90.000,E1 143.497} C_DIS
LIN {X 0.054,Y -628.542,Z 1279.594,A 0.000,B 0.000,C 90.000,E1 142.970} C_DIS
LIN {X -0.087,Y -631.075,Z 1279.592,A 0.000,B 0.000,C 90.000,E1 142.477} C_DIS
LIN {X -0.001,Y -635.718,Z 1279.586,A 0.000,B 0.000,C 90.000,E1 141.457} C_DIS
LIN {X -0.137,Y -637.839,Z 1279.583,A 0.000,B 0.000,C 90.000,E1 140.964} C_DIS
LIN {X 0.041,Y -640.811,Z 1279.579,A 0.000,B 0.000,C 90.000,E1 140.194} C_DIS
LIN {X -0.242,Y -644.549,Z 1279.573,A 0.000,B 0.000,C 90.000,E1 139.218} C_DIS
LIN {X -0.067,Y -648.935,Z 1279.566,A 0.000,B 0.000,C 90.000,E1 137.957} C_DIS
LIN {X 0.178,Y -652.192,Z 1279.561,A 0.000,B 0.000,C 90.000,E1 136.944} C_DIS
LIN {X -0.080,Y -656.975,Z 1279.553,A 0.000,B 0.000,C 90.000,E1 135.486} C_DIS
LIN {X -0.273,Y -663.466,Z 1279.542,A 0.000,B 0.000,C 90.000,E1 133.542} C_DIS
LIN {X 0.167,Y -667.498,Z 1279.535,A 0.000,B 0.000,C 90.000,E1 132.285} C_DIS
LIN {X 0.224,Y -670.678,Z 1279.530,A 0.000,B 0.000,C 90.000,E1 131.310} C_DIS
LIN {X -0.078,Y -675.280,Z 1279.522,A 0.000,B 0.000,C 90.000,E1 129.886} C_DIS
LIN {X 0.105,Y -678.878,Z 1279.515,A 0.000,B 0.000,C 90.000,E1 128.669} C_DIS
LIN {X -0.117,Y -681.626,Z 1279.510,A 0.000,B 0.000,C 90.000,E1 127.729} C_DIS
LIN {X 0.270,Y -684.894,Z 1279.503,A 0.000,B 0.000,C 90.000,E1 126.503} C_DIS
LIN {X 0.306,Y -687.855,Z 1279.496,A 0.000,B 0.000,C 90.000,E1 125.311} C_DIS
LIN {X 0.389,Y -690.637,Z 1279.490,A 0.000,B 0.000,C 90.000,E1 124.119} C_DIS
LIN {X -0.096,Y -692.594,Z 1279.484,A 0.000,B 0.000,C 90.000,E1 123.214} C_DIS
LIN {X 0.255,Y -694.857,Z 1279.478,A 0.000,B 0.000,C 90.000,E1 122.005} C_DIS
LIN {X 0.042,Y -696.481,Z 1279.473,A 0.000,B 0.000,C 90.000,E1 121.082} C_DIS
LIN {X -0.140,Y -698.362,Z 1279.466,A 0.000,B 0.000,C 90.000,E1 119.922} C_DIS
LIN {X -0.047,Y -699.996,Z 1279.460,A 0.000,B 0.000,C 90.000,E1 118.743} C_DIS
LIN {X 0.416,Y -701.020,Z 1279.454,A 0.000,B 0.000,C 90.000,E1 117.769} C_DIS
LIN {X -0.329,Y -701.636,Z 1279.451,A 0.000,B 0.000,C 90.000,E1 117.129} C_DIS
LIN {X 0.150,Y -701.876,Z 1279.445,A 0.000,B 0.000,C 90.000,E1 116.155} C_DIS
LIN {X -0.234,Y -701.835,Z 1279.443,A 0.000,B 0.000,C 90.000,E1 115.720} C_DIS
LIN {X -0.337,Y -701.429,Z 1279.439,A 0.000,B 0.000,C 90.000,E1 115.027} C_DIS
LIN {X -0.061,Y -701.232,Z 1279.438,A 0.000,B 0.000,C 90.000,E1 114.771} C_DIS
LIN {X 0.198,Y -700.535,Z 1279.435,A 0.000,B 0.000,C 90.000,E1 114.283} C_DIS
LIN {X -0.169,Y -700.065,Z 1279.434,A 0.000,B 0.000,C 90.000,E1 114.079} C_DIS
LIN {X 0.219,Y -697.734,Z 1279.431,A 0.000,B 0.000,C 90.000,E1 113.462} C_DIS
LIN {X -0.180,Y -694.229,Z 1279.428,A 0.000,B 0.000,C 90.000,E1 113.025} C_DIS
LIN {X -0.053,Y -693.285,Z 1279.427,A 0.000,B 0.000,C 90.000,E1 112.898} C_DIS
LIN {X 0.068,Y -691.901,Z 1279.427,A 0.000,B 0.000,C 90.000,E1 112.770} C_DIS
LIN {X 0.189,Y -689.716,Z 1279.426,A 0.000,B 0.000,C 90.000,E1 112.642} C_DIS
LIN {X -0.278,Y -685.831,Z 1279.425,A 0.000,B 0.000,C 90.000,E1 112.514} C_DIS
LIN {X 0.084,Y -683.982,Z 1279.424,A 0.000,B 0.000,C 90.000,E1 112.386} C_DIS
LIN {X -0.264,Y -681.907,Z 1279.424,A 0.000,B 0.000,C 90.000,E1 112.333} C_DIS
LIN {X 0.277,Y -679.172,Z 1279.424,A 0.000,B 0.000,C 90.000,E1 112.206} C_DIS
LIN {X 0.263,Y -669.644,Z 1279.423,A 0.000,B 0.000,C 90.000,E1 112.078} C_DIS
LIN {X 0.217,Y -665.292,Z 1279.423,A 0.000,B 0.000,C 90.000,E1 112.078} C_DIS
LIN {X 0.166,Y -638.438,Z 1279.423,A 0.000,B 0.000,C 90.000,E1 112.078} C_DIS
LIN {X -0.335,Y -635.856,Z 1279.422,A 0.000,B 0.000,C 90.000,E1 112.025} C_DIS
LIN {X 0.210,Y -635.821,Z 1279.422,A 0.000,B 0.000,C 90.000,E1 111.972} C_DIS
LIN {X -0.287,Y -636.642,Z 1279.421,A 0.000,B 0.000,C 90.000,E1 111.716} C_DIS
LIN {X 0.206,Y -641.456,Z 1279.417,A 0.000,B 0.000,C 90.000,E1 110.972} C_DIS
LIN {X 0.156,Y -645.123,Z 1279.414,A 0.000,B 0.000,C 90.000,E1 110.482} C_DIS
LIN {X -0.133,Y -649.363,Z 1279.410,A 0.000,B 0.000,C 90.000,E1 109.885} C_DIS
LIN {X -0.127,Y -653.643,Z 1279.406,A 0.000,B 0.000,C 90.000,E1 109.141} C_DIS
LIN {X -0.175,Y -656.188,Z 1279.404,A 0.000,B 0.000,C 90.000,E1 108.652} C_DIS
LIN {X 0.207,Y -658.582,Z 1279.401,A 0.000,B 0.000,C 90.000,E1 108.127} C_DIS
LIN {X 0.083,Y -661.882,Z 1279.397,A 0.000,B 0.000,C 90.000,E1 107.402} C_DIS
LIN {X 0.080,Y -663.936,Z 1279.394,A 0.000,B 0.000,C 90.000,E1 106.913} C_DIS
LIN {X -0.191,Y -666.628,Z 1279.390,A 0.000,B 0.000,C 90.000,E1 106.205} C_DIS
LIN {X -0.250,Y -668.845,Z 1279.386,A 0.000,B 0.000,C 90.000,E1 105.481} C_DIS
LIN {X 0.248,Y -670.197,Z 1279.383,A 0.000,B 0.000,C 90.000,E1 104.954} C_DIS
LIN {X 0.047,Y -671.697,Z 1279.379,A 0.000,B 0.000,C 90.000,E1 104.245} C_DIS
LIN {X -0.079,Y -672.490,Z 1279.376,A 0.000,B 0.000,C 90.000,E1 103.772} C_DIS
LIN {X -0.200,Y -673.119,Z 1279.374,A 0.000,B 0.000,C 90.000,E1 103.300} C_DIS
LIN {X 0.281,Y -673.633,Z 1279.370,A 0.000,B 0.000,C 90.000,E1 102.535} C_DIS
LIN {X 0.164,Y -673.784,Z 1279.367,A 0.000,B 0.000,C 90.000,E1 102.063} C_DIS
LIN {X 0.047,Y -673.744,Z 1279.365,A 0.000,B 0.000,C 90.000,E1 101.591} C_DIS
LIN {X -0.266,Y -673.244,Z 1279.360,A 0.000,B 0.000,C 90.000,E1 100.894} C_DIS
LIN {X 0.269,Y -672.754,Z 1279.358,A 0.000,B 0.000,C 90.000,E1 100.366} C_DIS
LIN {X 0.019,Y -671.909,Z 1279.355,A 0.000,B 0.000,C 90.000,E1 99.905} C_DIS
LIN {X -0.121,Y -670.851,Z 1279.352,A 0.000,B 0.000,C 90.000,E1 99.434} C_DIS
LIN {X 0.283,Y -669.524,Z 1279.350,A 0.000,B 0.000,C 90.000,E1 98.916} C_DIS
LIN {X 0.102,Y -668.757,Z 1279.348,A 0.000,B 0.000,C 90.000,E1 98.690} C_DIS
LIN {X -0.065,Y -666.950,Z 1279.346,A 0.000,B 0.000,C 90.000,E1 98.219} C_DIS
LIN {X 0.224,Y -664.226,Z 1279.342,A 0.000,B 0.000,C 90.000,E1 97.587} C_DIS
LIN {X -0.082,Y -660.946,Z 1279.339,A 0.000,B 0.000,C 90.000,E1 97.004} C_DIS
LIN {X 0.255,Y -657.993,Z 1279.336,A 0.000,B 0.000,C 90.000,E1 96.486} C_DIS
LIN {X -0.148,Y -654.669,Z 1279.333,A 0.000,B 0.000,C 90.000,E1 96.030} C_DIS
LIN {X 0.104,Y -650.058,Z 1279.330,A 0.000,B 0.000,C 90.000,E1 95.391} C_DIS
LIN {X -0.336,Y -646.034,Z 1279.327,A 0.000,B 0.000,C 90.000,E1 94.935} C_DIS
LIN {X -0.100,Y -641.559,Z 1279.325,A 0.000,B 0.000,C 90.000,E1 94.416} C_DIS
LIN {X 0.045,Y -635.490,Z 1279.321,A 0.000,B 0.000,C 90.000,E1 93.784} C_DIS
LIN {X -0.283,Y -630.464,Z 1279.318,A 0.000,B 0.000,C 90.000,E1 93.326} C_DIS
LIN {X 0.193,Y -625.226,Z 1279.316,A 0.000,B 0.000,C 90.000,E1 92.808} C_DIS
LIN {X 0.197,Y -615.383,Z 1279.311,A 0.000,B 0.000,C 90.000,E1 92.007} C_DIS
LIN {X -0.115,Y -609.618,Z 1279.309,A 0.000,B 0.000,C 90.000,E1 91.604} C_DIS
LIN {X -0.088,Y -601.928,Z 1279.306,A 0.000,B 0.000,C 90.000,E1 91.088} C_DIS
LIN {X 0.089,Y -595.654,Z 1279.304,A 0.000,B 0.000,C 90.000,E1 90.688} C_DIS
LIN {X 0.004,Y -588.638,Z 1279.302,A 0.000,B 0.000,C 90.000,E1 90.344} C_DIS
LIN {X -0.152,Y -581.298,Z 1279.300,A 0.000,B 0.000,C 90.000,E1 90.057} C_DIS
LIN {X 0.137,Y -576.203,Z 1279.299,A 0.000,B 0.000,C 90.000,E1 89.828} C_DIS
LIN {X -0.031,Y -572.406,Z 1279.298,A 0.000,B 0.000,C 90.000,E1 89.656} C_DIS
LIN {X 0.233,Y -571.253,Z 1279.298,A 0.000,B 0.000,C 90.000,E1 89.542} C_DIS
LIN {X 0.195,Y -570.571,Z 1279.297,A 0.000,B 0.000,C 90.000,E1 89.484} C_DIS
LIN {X -0.257,Y -569.397,Z 1279.296,A 0.000,B 0.000,C 90.000,E1 89.312} C_DIS
LIN {X -0.229,Y -568.954,Z 1279.293,A 0.000,B 0.000,C 90.000,E1 88.797} C_DIS
LIN {X -0.233,Y -571.987,Z 1279.272,A 0.000,B 0.000,C 90.000,E1 85.065} C_DIS
LIN {X -0.127,Y -574.344,Z 1279.260,A 0.000,B 0.000,C 90.000,E1 82.875} C_DIS
LIN {X -0.100,Y -576.573,Z 1279.250,A 0.000,B 0.000,C 90.000,E1 80.971} C_DIS
LIN {X 0.177,Y -577.738,Z 1279.244,A 0.000,B 0.000,C 90.000,E1 79.859} C_DIS
LIN {X -0.196,Y -578.764,Z 1279.238,A 0.000,B 0.000,C 90.000,E1 78.814} C_DIS
LIN {X 0.002,Y -580.173,Z 1279.229,A 0.000,B 0.000,C 90.000,E1 77.173} C_DIS
LIN {X -0.005,Y -581.299,Z 1279.221,A 0.000,B 0.000,C 90.000,E1 75.825} C_DIS
LIN {X 0.141,Y -582.252,Z 1279.214,A 0.000,B 0.000,C 90.000,E1 74.464} C_DIS
LIN {X -0.095,Y -583.082,Z 1279.206,A 0.000,B 0.000,C 90.000,E1 73.142} C_DIS
LIN {X -0.243,Y -584.352,Z 1279.196,A 0.000,B 0.000,C 90.000,E1 71.275} C_DIS
LIN {X -0.038,Y -585.168,Z 1279.187,A 0.000,B 0.000,C 90.000,E1 69.645} C_DIS
LIN {X -0.007,Y -586.565,Z 1279.174,A 0.000,B 0.000,C 90.000,E1 67.230} C_DIS
LIN {X 0.000,Y -588.000,Z 1279.163,A 0.000,B 0.000,C 90.000,E1 65.357} C_DIS
LIN {X -0.138,Y -589.239,Z 1279.154,A 0.000,B 0.000,C 90.000,E1 63.768} C_DIS
LIN {X -0.089,Y -590.838,Z 1279.144,A 0.000,B 0.000,C 90.000,E1 61.897} C_DIS
LIN {X 0.089,Y -592.419,Z 1279.135,A 0.000,B 0.000,C 90.000,E1 60.284} C_DIS
LIN {X -0.235,Y -594.349,Z 1279.125,A 0.000,B 0.000,C 90.000,E1 58.456} C_DIS
LIN {X -0.117,Y -595.697,Z 1279.117,A 0.000,B 0.000,C 90.000,E1 57.120} C_DIS
LIN {X -0.381,Y -596.810,Z 1279.111,A 0.000,B 0.000,C 90.000,E1 56.087} C_DIS
LIN {X -0.166,Y -598.384,Z 1279.103,A 0.000,B 0.000,C 90.000,E1 54.482} C_DIS
LIN {X -0.046,Y -599.757,Z 1279.094,A 0.000,B 0.000,C 90.000,E1 52.889} C_DIS
LIN {X -0.020,Y -601.242,Z 1279.084,A 0.000,B 0.000,C 90.000,E1 51.045} C_DIS
LIN {X -0.213,Y -601.764,Z 1279.079,A 0.000,B 0.000,C 90.000,E1 50.275} C_DIS
LIN {X 0.065,Y -602.157,Z 1279.075,A 0.000,B 0.000,C 90.000,E1 49.461} C_DIS
LIN {X 0.168,Y -602.838,Z 1279.066,A 0.000,B 0.000,C 90.000,E1 47.877} C_DIS
LIN {X 0.206,Y -603.225,Z 1279.060,A 0.000,B 0.000,C 90.000,E1 46.824} C_DIS
LIN {X -0.358,Y -603.458,Z 1279.053,A 0.000,B 0.000,C 90.000,E1 45.567} C_DIS
LIN {X 0.352,Y -603.415,Z 1279.046,A 0.000,B 0.000,C 90.000,E1 44.190} C_DIS
LIN {X -0.212,Y -603.115,Z 1279.038,A 0.000,B 0.000,C 90.000,E1 42.933} C_DIS
LIN {X 0.067,Y -602.709,Z 1279.031,A 0.000,B 0.000,C 90.000,E1 41.595} C_DIS
LIN {X 0.142,Y -602.228,Z 1279.025,A 0.000,B 0.000,C 90.000,E1 40.539} C_DIS
LIN {X -0.036,Y -601.884,Z 1279.021,A 0.000,B 0.000,C 90.000,E1 39.769} C_DIS
LIN {X -0.139,Y -601.465,Z 1279.017,A 0.000,B 0.000,C 90.000,E1 38.991} C_DIS
LIN {X 0.138,Y -600.938,Z 1279.012,A 0.000,B 0.000,C 90.000,E1 38.177} C_DIS
LIN {X -0.191,Y -600.010,Z 1279.006,A 0.000,B 0.000,C 90.000,E1 37.156} C_DIS
LIN {X -0.055,Y -598.727,Z 1279.000,A 0.000,B 0.000,C 90.000,E1 36.091} C_DIS
LIN {X 0.061,Y -597.293,Z 1278.995,A 0.000,B 0.000,C 90.000,E1 35.025} C_DIS
LIN {X 0.038,Y -594.901,Z 1278.987,A 0.000,B 0.000,C 90.000,E1 33.706} C_DIS
LIN {X 0.150,Y -593.910,Z 1278.984,A 0.000,B 0.000,C 90.000,E1 33.166} C_DIS
LIN {X -0.350,Y -592.058,Z 1278.980,A 0.000,B 0.000,C 90.000,E1 32.418} C_DIS
LIN {X -0.168,Y -589.146,Z 1278.974,A 0.000,B 0.000,C 90.000,E1 31.337} C_DIS
LIN {X -0.210,Y -586.613,Z 1278.970,A 0.000,B 0.000,C 90.000,E1 30.541} C_DIS
LIN {X -0.154,Y -584.740,Z 1278.967,A 0.000,B 0.000,C 90.000,E1 30.001} C_DIS
LIN {X -0.244,Y -581.456,Z 1278.962,A 0.000,B 0.000,C 90.000,E1 29.205} C_DIS
LIN {X 0.208,Y -578.436,Z 1278.958,A 0.000,B 0.000,C 90.000,E1 28.487} C_DIS
LIN {X -0.006,Y -576.411,Z 1278.956,A 0.000,B 0.000,C 90.000,E1 28.103} C_DIS
LIN {X 0.312,Y -572.107,Z 1278.952,A 0.000,B 0.000,C 90.000,E1 27.257} C_DIS
LIN {X -0.187,Y -567.295,Z 1278.947,A 0.000,B 0.000,C 90.000,E1 26.488} C_DIS
LIN {X -0.128,Y -562.910,Z 1278.943,A 0.000,B 0.000,C 90.000,E1 25.796} C_DIS
LIN {X 0.134,Y -558.174,Z 1278.939,A 0.000,B 0.000,C 90.000,E1 25.079} C_DIS
LIN {X 0.219,Y -554.123,Z 1278.936,A 0.000,B 0.000,C 90.000,E1 24.515} C_DIS
LIN {X 0.157,Y -548.678,Z 1278.932,A 0.000,B 0.000,C 90.000,E1 23.823} C_DIS
LIN {X -0.064,Y -541.746,Z 1278.928,A 0.000,B 0.000,C 90.000,E1 23.025} C_DIS
LIN {X -0.177,Y -535.493,Z 1278.924,A 0.000,B 0.000,C 90.000,E1 22.333} C_DIS
LIN {X 0.143,Y -527.743,Z 1278.919,A 0.000,B 0.000,C 90.000,E1 21.461} C_DIS
LIN {X -0.120,Y -519.866,Z 1278.915,A 0.000,B 0.000,C 90.000,E1 20.663} C_DIS
LIN {X -0.108,Y -514.678,Z 1278.912,A 0.000,B 0.000,C 90.000,E1 20.120} C_DIS
LIN {X 0.074,Y -503.970,Z 1278.906,A 0.000,B 0.000,C 90.000,E1 19.033} C_DIS
LIN {X -0.268,Y -492.843,Z 1278.900,A 0.000,B 0.000,C 90.000,E1 18.000} C_DIS
LIN {X 0.117,Y -485.617,Z 1278.896,A 0.000,B 0.000,C 90.000,E1 17.275} C_DIS
LIN {X -0.026,Y -476.735,Z 1278.892,A 0.000,B 0.000,C 90.000,E1 16.496} C_DIS
LIN {X 0.131,Y -466.371,Z 1278.887,A 0.000,B 0.000,C 90.000,E1 15.552} C_DIS
LIN {X 0.063,Y -448.700,Z 1278.878,A 0.000,B 0.000,C 90.000,E1 13.953} C_DIS
LIN {X 0.076,Y -425.440,Z 1278.865,A 0.000,B 0.000,C 90.000,E1 11.658} C_DIS
LIN {X 0.141,Y -409.664,Z 1278.855,A 0.000,B 0.000,C 90.000,E1 9.962} C_DIS
LIN {X -0.193,Y -399.963,Z 1278.849,A 0.000,B 0.000,C 90.000,E1 8.916} C_DIS
LIN {X -0.104,Y -396.310,Z 1278.847,A 0.000,B 0.000,C 90.000,E1 8.398} C_DIS
LIN {X 0.100,Y -394.963,Z 1278.845,A 0.000,B 0.000,C 90.000,E1 8.106} C_DIS
LIN {X 0.062,Y -394.941,Z 1278.845,A 0.000,B 0.000,C 90.000,E1 8.106} C_DIS
LIN {X 0.025,Y -394.938,Z 1278.845,A 0.000,B 0.000,C 90.000,E1 8.106} C_DIS
LIN {X -0.107,Y -395.162,Z 1278.845,A 0.000,B 0.000,C 90.000,E1 8.049} C_DIS
LIN {X -0.097,Y -396.296,Z 1278.844,A 0.000,B 0.000,C 90.000,E1 7.871} C_DIS
LIN {X 0.025,Y -399.747,Z 1278.842,A 0.000,B 0.000,C 90.000,E1 7.530} C_DIS
LIN {X -0.023,Y -410.745,Z 1278.838,A 0.000,B 0.000,C 90.000,E1 6.891} C_DIS
LIN {X -0.141,Y -417.291,Z 1278.836,A 0.000,B 0.000,C 90.000,E1 6.486} C_DIS
LIN {X -0.134,Y -425.193,Z 1278.833,A 0.000,B 0.000,C 90.000,E1 5.910} C_DIS
LIN {X 0.005,Y -433.144,Z 1278.829,A 0.000,B 0.000,C 90.000,E1 5.277} C_DIS
LIN {X 0.000,Y -442.510,Z 1278.825,A 0.000,B 0.000,C 90.000,E1 4.531} C_DIS
LIN {X -0.130,Y -453.049,Z 1278.820,A 0.000,B 0.000,C 90.000,E1 3.669} C_DIS
LIN {X 0.096,Y -460.460,Z 1278.817,A 0.000,B 0.000,C 90.000,E1 2.980} C_DIS
LIN {X 0.130,Y -467.424,Z 1278.813,A 0.000,B 0.000,C 90.000,E1 2.293} C_DIS
LIN {X 0.088,Y -473.031,Z 1278.810,A 0.000,B 0.000,C 90.000,E1 1.718} C_DIS
LIN {X 0.128,Y -479.658,Z 1278.806,A 0.000,B 0.000,C 90.000,E1 0.974} C_DIS
LIN {X -0.067,Y -485.955,Z 1278.801,A 0.000,B 0.000,C 90.000,E1 0.229} C_DIS
LIN {X 0.019,Y -491.550,Z 1278.797,A 0.000,B 0.000,C 90.000,E1 359.484} C_DIS
LIN {X 0.062,Y -497.774,Z 1278.792,A 0.000,B 0.000,C 90.000,E1 358.568} C_DIS
LIN {X 0.002,Y -502.573,Z 1278.788,A 0.000,B 0.000,C 90.000,E1 357.822} C_DIS
LIN {X -0.035,Y -507.073,Z 1278.784,A 0.000,B 0.000,C 90.000,E1 357.078} C_DIS
LIN {X -0.213,Y -510.505,Z 1278.781,A 0.000,B 0.000,C 90.000,E1 356.502} C_DIS
LIN {X -0.150,Y -514.474,Z 1278.776,A 0.000,B 0.000,C 90.000,E1 355.755} C_DIS
LIN {X 0.246,Y -517.476,Z 1278.773,A 0.000,B 0.000,C 90.000,E1 355.122} C_DIS
LIN {X 0.078,Y -523.022,Z 1278.767,A 0.000,B 0.000,C 90.000,E1 353.970} C_DIS
LIN {X 0.255,Y -526.132,Z 1278.763,A 0.000,B 0.000,C 90.000,E1 353.223} C_DIS
LIN {X 0.237,Y -529.501,Z 1278.758,A 0.000,B 0.000,C 90.000,E1 352.356} C_DIS
LIN {X 0.253,Y -532.671,Z 1278.753,A 0.000,B 0.000,C 90.000,E1 351.489} C_DIS
LIN {X -0.228,Y -535.531,Z 1278.748,A 0.000,B 0.000,C 90.000,E1 350.679} C_DIS
LIN {X -0.062,Y -538.087,Z 1278.743,A 0.000,B 0.000,C 90.000,E1 349.803} C_DIS
LIN {X 0.138,Y -540.436,Z 1278.739,A 0.000,B 0.000,C 90.000,E1 348.926} C_DIS
LIN {X -0.165,Y -542.480,Z 1278.734,A 0.000,B 0.000,C 90.000,E1 348.105} C_DIS
LIN {X 0.084,Y -544.479,Z 1278.729,A 0.000,B 0.000,C 90.000,E1 347.229} C_DIS
LIN {X -0.180,Y -546.273,Z 1278.724,A 0.000,B 0.000,C 90.000,E1 346.408} C_DIS
LIN {X 0.004,Y -547.296,Z 1278.721,A 0.000,B 0.000,C 90.000,E1 345.825} C_DIS
LIN {X -0.007,Y -549.115,Z 1278.715,A 0.000,B 0.000,C 90.000,E1 344.700} C_DIS
LIN {X -0.093,Y -550.259,Z 1278.710,A 0.000,B 0.000,C 90.000,E1 343.866} C_DIS
LIN {X 0.093,Y -551.492,Z 1278.704,A 0.000,B 0.000,C 90.000,E1 342.725} C_DIS
LIN {X 0.200,Y -552.168,Z 1278.699,A 0.000,B 0.000,C 90.000,E1 341.873} C_DIS
LIN {X 0.047,Y -552.495,Z 1278.696,A 0.000,B 0.000,C 90.000,E1 341.329} C_DIS
LIN {X -0.105,Y -552.674,Z 1278.693,A 0.000,B 0.000,C 90.000,E1 340.786} C_DIS
LIN {X 0.021,Y -552.556,Z 1278.689,A 0.000,B 0.000,C 90.000,E1 339.934} C_DIS
LIN {X 0.145,Y -552.129,Z 1278.684,A 0.000,B 0.000,C 90.000,E1 339.082} C_DIS
LIN {X -0.254,Y -551.505,Z 1278.679,A 0.000,B 0.000,C 90.000,E1 338.284} C_DIS
LIN {X 0.294,Y -550.829,Z 1278.676,A 0.000,B 0.000,C 90.000,E1 337.667} C_DIS
LIN {X -0.123,Y -549.635,Z 1278.672,A 0.000,B 0.000,C 90.000,E1 336.869} C_DIS
LIN {X -0.320,Y -547.079,Z 1278.664,A 0.000,B 0.000,C 90.000,E1 335.485} C_DIS
LIN {X -0.080,Y -545.893,Z 1278.661,A 0.000,B 0.000,C 90.000,E1 334.897} C_DIS
LIN {X 0.164,Y -543.638,Z 1278.656,A 0.000,B 0.000,C 90.000,E1 334.024} C_DIS
LIN {X -0.114,Y -541.222,Z 1278.651,A 0.000,B 0.000,C 90.000,E1 333.204} C_DIS
LIN {X -0.172,Y -538.304,Z 1278.646,A 0.000,B 0.000,C 90.000,E1 332.359} C_DIS
LIN {X -0.258,Y -535.050,Z 1278.642,A 0.000,B 0.000,C 90.000,E1 331.513} C_DIS
LIN {X -0.093,Y -532.644,Z 1278.638,A 0.000,B 0.000,C 90.000,E1 330.923} C_DIS
LIN {X 0.049,Y -530.003,Z 1278.635,A 0.000,B 0.000,C 90.000,E1 330.333} C_DIS
LIN {X 0.016,Y -526.263,Z 1278.631,A 0.000,B 0.000,C 90.000,E1 329.616} C_DIS
LIN {X -0.171,Y -518.825,Z 1278.624,A 0.000,B 0.000,C 90.000,E1 328.329} C_DIS
LIN {X -0.040,Y -511.213,Z 1278.617,A 0.000,B 0.000,C 90.000,E1 326.993} C_DIS
LIN {X 0.110,Y -506.817,Z 1278.612,A 0.000,B 0.000,C 90.000,E1 326.087} C_DIS
LIN {X -0.183,Y -504.890,Z 1278.609,A 0.000,B 0.000,C 90.000,E1 325.674} C_DIS
LIN {X -0.135,Y -502.837,Z 1278.606,A 0.000,B 0.000,C 90.000,E1 325.102} C_DIS
LIN {X -0.021,Y -500.932,Z 1278.602,A 0.000,B 0.000,C 90.000,E1 324.276} C_DIS
LIN {X 0.021,Y -499.422,Z 1278.597,A 0.000,B 0.000,C 90.000,E1 323.371} C_DIS
LIN {X -0.182,Y -498.455,Z 1278.590,A 0.000,B 0.000,C 90.000,E1 322.190} C_DIS
LIN {X 0.050,Y -498.060,Z 1278.580,A 0.000,B 0.000,C 90.000,E1 320.356} C_DIS
LIN {X 0.160,Y -498.194,Z 1278.573,A 0.000,B 0.000,C 90.000,E1 319.138} C_DIS
LIN {X 0.134,Y -498.409,Z 1278.565,A 0.000,B 0.000,C 90.000,E1 317.634} C_DIS
LIN {X 0.274,Y -498.691,Z 1278.555,A 0.000,B 0.000,C 90.000,E1 315.810} C_DIS
LIN {X 0.065,Y -499.052,Z 1278.545,A 0.000,B 0.000,C 90.000,E1 314.028} C_DIS
LIN {X 0.081,Y -499.438,Z 1278.533,A 0.000,B 0.000,C 90.000,E1 311.919} C_DIS
LIN {X 0.279,Y -499.780,Z 1278.523,A 0.000,B 0.000,C 90.000,E1 310.092} C_DIS
LIN {X 0.154,Y -500.026,Z 1278.513,A 0.000,B 0.000,C 90.000,E1 308.302} C_DIS
LIN {X 0.059,Y -500.154,Z 1278.506,A 0.000,B 0.000,C 90.000,E1 307.111} C_DIS
LIN {X 0.151,Y -500.189,Z 1278.498,A 0.000,B 0.000,C 90.000,E1 305.598} C_DIS
LIN {X 0.190,Y -499.901,Z 1278.493,A 0.000,B 0.000,C 90.000,E1 304.692} C_DIS
LIN {X 0.226,Y -499.254,Z 1278.488,A 0.000,B 0.000,C 90.000,E1 303.785} C_DIS
LIN {X -0.033,Y -498.493,Z 1278.484,A 0.000,B 0.000,C 90.000,E1 303.214} C_DIS
LIN {X -0.153,Y -497.415,Z 1278.481,A 0.000,B 0.000,C 90.000,E1 302.625} C_DIS
LIN {X 0.131,Y -496.687,Z 1278.479,A 0.000,B 0.000,C 90.000,E1 302.291} C_DIS
LIN {X -0.010,Y -495.722,Z 1278.478,A 0.000,B 0.000,C 90.000,E1 302.005} C_DIS
LIN {X -0.154,Y -494.231,Z 1278.476,A 0.000,B 0.000,C 90.000,E1 301.720} C_DIS
LIN {X -0.189,Y -479.614,Z 1278.460,A 0.000,B 0.000,C 90.000,E1 298.821} C_DIS
LIN {X -0.104,Y -466.776,Z 1278.444,A 0.000,B 0.000,C 90.000,E1 295.848} C_DIS
LIN {X 0.138,Y -455.092,Z 1278.426,A 0.000,B 0.000,C 90.000,E1 292.642} C_DIS
LIN {X -0.147,Y -445.187,Z 1278.408,A 0.000,B 0.000,C 90.000,E1 289.450} C_DIS
LIN {X -0.132,Y -436.251,Z 1278.388,A 0.000,B 0.000,C 90.000,E1 285.843} C_DIS
LIN {X 0.207,Y -428.230,Z 1278.364,A 0.000,B 0.000,C 90.000,E1 281.478} C_DIS
LIN {X -0.134,Y -421.994,Z 1278.334,A 0.000,B 0.000,C 90.000,E1 276.144} C_DIS
LIN {X -0.132,Y -423.408,Z 1278.259,A 0.000,B 0.000,C 90.000,E1 262.591} C_DIS
LIN {X -0.107,Y -429.672,Z 1278.233,A 0.000,B 0.000,C 90.000,E1 257.881} C_DIS
LIN {X 0.082,Y -437.518,Z 1278.210,A 0.000,B 0.000,C 90.000,E1 253.866} C_DIS
LIN {X 0.185,Y -446.800,Z 1278.190,A 0.000,B 0.000,C 90.000,E1 250.242} C_DIS
LIN {X -0.148,Y -457.051,Z 1278.172,A 0.000,B 0.000,C 90.000,E1 247.050} C_DIS
LIN {X 0.119,Y -464.063,Z 1278.162,A 0.000,B 0.000,C 90.000,E1 245.101} C_DIS
LIN {X 0.046,Y -465.004,Z 1278.160,A 0.000,B 0.000,C 90.000,E1 244.793} C_DIS
LIN {X 0.173,Y -465.584,Z 1278.158,A 0.000,B 0.000,C 90.000,E1 244.460} C_DIS
LIN {X 0.036,Y -466.255,Z 1278.155,A 0.000,B 0.000,C 90.000,E1 243.845} C_DIS
LIN {X 0.250,Y -466.661,Z 1278.150,A 0.000,B 0.000,C 90.000,E1 242.871} C_DIS
LIN {X -0.158,Y -466.651,Z 1278.144,A 0.000,B 0.000,C 90.000,E1 241.975} C_DIS
LIN {X -0.197,Y -466.296,Z 1278.137,A 0.000,B 0.000,C 90.000,E1 240.717} C_DIS
LIN {X -0.086,Y -465.507,Z 1278.128,A 0.000,B 0.000,C 90.000,E1 239.125} C_DIS
LIN {X -0.251,Y -464.304,Z 1278.118,A 0.000,B 0.000,C 90.000,E1 237.248} C_DIS
LIN {X 0.058,Y -463.078,Z 1278.107,A 0.000,B 0.000,C 90.000,E1 235.308} C_DIS
LIN {X 0.101,Y -461.670,Z 1278.093,A 0.000,B 0.000,C 90.000,E1 232.763} C_DIS
LIN {X -0.130,Y -460.799,Z 1278.083,A 0.000,B 0.000,C 90.000,E1 230.884} C_DIS
LIN {X 0.198,Y -460.096,Z 1278.072,A 0.000,B 0.000,C 90.000,E1 228.933} C_DIS
LIN {X -0.179,Y -459.501,Z 1278.061,A 0.000,B 0.000,C 90.000,E1 227.067} C_DIS
LIN {X -0.172,Y -458.951,Z 1278.047,A 0.000,B 0.000,C 90.000,E1 224.514} C_DIS
LIN {X 0.063,Y -459.163,Z 1278.024,A 0.000,B 0.000,C 90.000,E1 220.334} C_DIS
LIN {X -0.023,Y -459.527,Z 1278.015,A 0.000,B 0.000,C 90.000,E1 218.749} C_DIS
LIN {X -0.053,Y -463.955,Z 1277.980,A 0.000,B 0.000,C 90.000,E1 212.388} C_DIS
LIN {X -0.101,Y -466.596,Z 1277.968,A 0.000,B 0.000,C 90.000,E1 210.178} C_DIS
LIN {X -0.061,Y -468.761,Z 1277.957,A 0.000,B 0.000,C 90.000,E1 208.281} C_DIS
LIN {X -0.084,Y -471.966,Z 1277.943,A 0.000,B 0.000,C 90.000,E1 205.771} C_DIS
LIN {X 0.013,Y -475.589,Z 1277.929,A 0.000,B 0.000,C 90.000,E1 203.259} C_DIS
LIN {X -0.130,Y -479.099,Z 1277.917,A 0.000,B 0.000,C 90.000,E1 201.099} C_DIS
LIN {X -0.053,Y -484.358,Z 1277.900,A 0.000,B 0.000,C 90.000,E1 198.000} C_DIS
LIN {X 0.147,Y -487.710,Z 1277.890,A 0.000,B 0.000,C 90.000,E1 196.134} C_DIS
LIN {X 0.266,Y -490.495,Z 1277.881,A 0.000,B 0.000,C 90.000,E1 194.592} C_DIS
LIN {X 0.124,Y -494.497,Z 1277.870,A 0.000,B 0.000,C 90.000,E1 192.479} C_DIS
LIN {X 0.257,Y -497.414,Z 1277.861,A 0.000,B 0.000,C 90.000,E1 190.950} C_DIS
LIN {X 0.180,Y -500.824,Z 1277.851,A 0.000,B 0.000,C 90.000,E1 189.151} C_DIS
LIN {X 0.181,Y -504.409,Z 1277.841,A 0.000,B 0.000,C 90.000,E1 187.352} C_DIS
LIN {X -0.198,Y -506.715,Z 1277.834,A 0.000,B 0.000,C 90.000,E1 186.201} C_DIS
LIN {X -0.197,Y -510.006,Z 1277.824,A 0.000,B 0.000,C 90.000,E1 184.416} C_DIS
LIN {X -0.022,Y -512.278,Z 1277.818,A 0.000,B 0.000,C 90.000,E1 183.212} C_DIS
LIN {X 0.133,Y -514.926,Z 1277.810,A 0.000,B 0.000,C 90.000,E1 181.718} C_DIS
LIN {X -0.216,Y -517.443,Z 1277.802,A 0.000,B 0.000,C 90.000,E1 180.286} C_DIS
LIN {X -0.057,Y -520.344,Z 1277.792,A 0.000,B 0.000,C 90.000,E1 178.511} C_DIS
LIN {X -0.250,Y -522.100,Z 1277.785,A 0.000,B 0.000,C 90.000,E1 177.364} C_DIS
LIN {X 0.095,Y -524.050,Z 1277.777,A 0.000,B 0.000,C 90.000,E1 175.869} C_DIS
LIN {X -0.047,Y -525.360,Z 1277.771,A 0.000,B 0.000,C 90.000,E1 174.723} C_DIS
LIN {X -0.117,Y -526.758,Z 1277.763,A 0.000,B 0.000,C 90.000,E1 173.280} C_DIS
LIN {X -0.139,Y -527.977,Z 1277.753,A 0.000,B 0.000,C 90.000,E1 171.546} C_DIS
LIN {X -0.116,Y -528.425,Z 1277.747,A 0.000,B 0.000,C 90.000,E1 170.387} C_DIS
LIN {X 0.004,Y -528.673,Z 1277.740,A 0.000,B 0.000,C 90.000,E1 169.218} C_DIS
LIN {X 0.131,Y -528.676,Z 1277.734,A 0.000,B 0.000,C 90.000,E1 168.049} C_DIS
LIN {X -0.233,Y -528.324,Z 1277.726,A 0.000,B 0.000,C 90.000,E1 166.645} C_DIS
LIN {X 0.023,Y -527.811,Z 1277.718,A 0.000,B 0.000,C 90.000,E1 165.172} C_DIS
LIN {X -0.242,Y -526.863,Z 1277.702,A 0.000,B 0.000,C 90.000,E1 162.308} C_DIS
LIN {X 0.098,Y -526.790,Z 1277.697,A 0.000,B 0.000,C 90.000,E1 161.402} C_DIS
LIN {X -0.213,Y -527.362,Z 1277.687,A 0.000,B 0.000,C 90.000,E1 159.699} C_DIS
LIN {X -0.175,Y -528.277,Z 1277.682,A 0.000,B 0.000,C 90.000,E1 158.827} C_DIS
LIN {X 0.173,Y -529.697,Z 1277.677,A 0.000,B 0.000,C 90.000,E1 157.922} C_DIS
LIN {X 0.053,Y -530.983,Z 1277.674,A 0.000,B 0.000,C 90.000,E1 157.358} C_DIS
LIN {X 0.136,Y -533.313,Z 1277.670,A 0.000,B 0.000,C 90.000,E1 156.485} C_DIS
LIN {X -0.099,Y -536.072,Z 1277.666,A 0.000,B 0.000,C 90.000,E1 155.793} C_DIS
LIN {X 0.179,Y -539.335,Z 1277.661,A 0.000,B 0.000,C 90.000,E1 155.049} C_DIS
LIN {X -0.227,Y -541.616,Z 1277.659,A 0.000,B 0.000,C 90.000,E1 154.665} C_DIS
LIN {X 0.103,Y -544.238,Z 1277.657,A 0.000,B 0.000,C 90.000,E1 154.204} C_DIS
LIN {X -0.156,Y -551.153,Z 1277.651,A 0.000,B 0.000,C 90.000,E1 153.256} C_DIS
LIN {X 0.015,Y -556.833,Z 1277.647,A 0.000,B 0.000,C 90.000,E1 152.538} C_DIS
LIN {X -0.005,Y -569.057,Z 1277.640,A 0.000,B 0.000,C 90.000,E1 151.179} C_DIS
LIN {X -0.302,Y -580.156,Z 1277.633,A 0.000,B 0.000,C 90.000,E1 149.999} C_DIS
LIN {X 0.356,Y -588.638,Z 1277.628,A 0.000,B 0.000,C 90.000,E1 148.997} C_DIS
LIN {X 0.117,Y -593.336,Z 1277.625,A 0.000,B 0.000,C 90.000,E1 148.486} C_DIS
LIN {X -0.067,Y -599.998,Z 1277.621,A 0.000,B 0.000,C 90.000,E1 147.709} C_DIS
LIN {X 0.084,Y -604.144,Z 1277.618,A 0.000,B 0.000,C 90.000,E1 147.168} C_DIS
LIN {X 0.231,Y -609.003,Z 1277.614,A 0.000,B 0.000,C 90.000,E1 146.501} C_DIS
LIN {X -0.095,Y -613.646,Z 1277.610,A 0.000,B 0.000,C 90.000,E1 145.881} C_DIS
LIN {X -0.034,Y -617.768,Z 1277.607,A 0.000,B 0.000,C 90.000,E1 145.229} C_DIS
LIN {X 0.217,Y -621.607,Z 1277.603,A 0.000,B 0.000,C 90.000,E1 144.562} C_DIS
LIN {X 0.136,Y -624.440,Z 1277.600,A 0.000,B 0.000,C 90.000,E1 144.069} C_DIS
LIN {X 0.021,Y -629.122,Z 1277.596,A 0.000,B 0.000,C 90.000,E1 143.210} C_DIS
LIN {X 0.088,Y -633.278,Z 1277.591,A 0.000,B 0.000,C 90.000,E1 142.316} C_DIS
LIN {X 0.321,Y -636.628,Z 1277.587,A 0.000,B 0.000,C 90.000,E1 141.537} C_DIS
LIN {X -0.305,Y -638.701,Z 1277.584,A 0.000,B 0.000,C 90.000,E1 141.090} C_DIS
LIN {X -0.217,Y -643.405,Z 1277.577,A 0.000,B 0.000,C 90.000,E1 139.828} C_DIS
LIN {X 0.016,Y -646.882,Z 1277.571,A 0.000,B 0.000,C 90.000,E1 138.809} C_DIS
LIN {X 0.172,Y -651.085,Z 1277.564,A 0.000,B 0.000,C 90.000,E1 137.553} C_DIS
LIN {X 0.330,Y -656.501,Z 1277.555,A 0.000,B 0.000,C 90.000,E1 135.810} C_DIS
LIN {X 0.145,Y -662.012,Z 1277.545,A 0.000,B 0.000,C 90.000,E1 134.109} C_DIS
LIN {X 0.089,Y -665.261,Z 1277.540,A 0.000,B 0.000,C 90.000,E1 133.137} C_DIS
LIN {X 0.113,Y -670.007,Z 1277.532,A 0.000,B 0.000,C 90.000,E1 131.676} C_DIS
LIN {X -0.208,Y -674.553,Z 1277.524,A 0.000,B 0.000,C 90.000,E1 130.253} C_DIS
LIN {X -0.073,Y -676.768,Z 1277.520,A 0.000,B 0.000,C 90.000,E1 129.519} C_DIS
LIN {X 0.131,Y -680.268,Z 1277.513,A 0.000,B 0.000,C 90.000,E1 128.302} C_DIS
LIN {X -0.073,Y -682.943,Z 1277.508,A 0.000,B 0.000,C 90.000,E1 127.363} C_DIS
LIN {X 0.306,Y -685.481,Z 1277.502,A 0.000,B 0.000,C 90.000,E1 126.377} C_DIS
LIN {X -0.206,Y -688.417,Z 1277.496,A 0.000,B 0.000,C 90.000,E1 125.231} C_DIS
LIN {X -0.146,Y -690.621,Z 1277.490,A 0.000,B 0.000,C 90.000,E1 124.278} C_DIS
LIN {X -0.023,Y -693.042,Z 1277.484,A 0.000,B 0.000,C 90.000,E1 123.086} C_DIS
LIN {X -0.250,Y -695.311,Z 1277.477,A 0.000,B 0.000,C 90.000,E1 121.926} C_DIS
LIN {X -0.462,Y -696.948,Z 1277.472,A 0.000,B 0.000,C 90.000,E1 121.003} C_DIS
LIN {X 0.308,Y -698.483,Z 1277.467,A 0.000,B 0.000,C 90.000,E1 120.001} C_DIS
LIN {X -0.204,Y -700.149,Z 1277.460,A 0.000,B 0.000,C 90.000,E1 118.871} C_DIS
LIN {X 0.259,Y -701.189,Z 1277.455,A 0.000,B 0.000,C 90.000,E1 117.897} C_DIS
LIN {X -0.207,Y -702.036,Z 1277.450,A 0.000,B 0.000,C 90.000,E1 117.001} C_DIS
LIN {X -0.032,Y -702.216,Z 1277.445,A 0.000,B 0.000,C 90.000,E1 116.052} C_DIS
LIN {X -0.105,Y -702.119,Z 1277.442,A 0.000,B 0.000,C 90.000,E1 115.591} C_DIS
LIN {X -0.206,Y -701.678,Z 1277.438,A 0.000,B 0.000,C 90.000,E1 114.899} C_DIS
LIN {X 0.070,Y -701.449,Z 1277.437,A 0.000,B 0.000,C 90.000,E1 114.643} C_DIS
LIN {X -0.309,Y -700.732,Z 1277.434,A 0.000,B 0.000,C 90.000,E1 114.207} C_DIS
LIN {X -0.037,Y -700.006,Z 1277.433,A 0.000,B 0.000,C 90.000,E1 113.951} C_DIS
LIN {X 0.219,Y -698.128,Z 1277.431,A 0.000,B 0.000,C 90.000,E1 113.462} C_DIS
LIN {X -0.158,Y -696.437,Z 1277.429,A 0.000,B 0.000,C 90.000,E1 113.259} C_DIS
LIN {X -0.001,Y -693.732,Z 1277.427,A 0.000,B 0.000,C 90.000,E1 112.898} C_DIS
LIN {X 0.123,Y -692.427,Z 1277.427,A 0.000,B 0.000,C 90.000,E1 112.770} C_DIS
LIN {X 0.309,Y -690.460,Z 1277.426,A 0.000,B 0.000,C 90.000,E1 112.642} C_DIS
LIN {X 0.081,Y -682.903,Z 1277.424,A 0.000,B 0.000,C 90.000,E1 112.333} C_DIS
LIN {X 0.141,Y -678.806,Z 1277.423,A 0.000,B 0.000,C 90.000,E1 112.206} C_DIS
LIN {X 0.131,Y -674.570,Z 1277.423,A 0.000,B 0.000,C 90.000,E1 112.153} C_DIS
LIN {X 0.120,Y -670.015,Z 1277.423,A 0.000,B 0.000,C 90.000,E1 112.099} C_DIS
LIN {X 0.066,Y -637.891,Z 1277.423,A 0.000,B 0.000,C 90.000,E1 112.099} C_DIS
LIN {X -0.239,Y -635.166,Z 1277.422,A 0.000,B 0.000,C 90.000,E1 112.025} C_DIS
LIN {X -0.281,Y -635.068,Z 1277.422,A 0.000,B 0.000,C 90.000,E1 112.025} C_DIS
LIN {X -0.077,Y -635.903,Z 1277.421,A 0.000,B 0.000,C 90.000,E1 111.716} C_DIS
LIN {X -0.246,Y -636.667,Z 1277.420,A 0.000,B 0.000,C 90.000,E1 111.589} C_DIS
LIN {X 0.184,Y -643.384,Z 1277.415,A 0.000,B 0.000,C 90.000,E1 110.610} C_DIS
LIN {X 0.105,Y -647.736,Z 1277.411,A 0.000,B 0.000,C 90.000,E1 109.993} C_DIS
LIN {X 0.020,Y -650.702,Z 1277.408,A 0.000,B 0.000,C 90.000,E1 109.504} C_DIS
LIN {X -0.220,Y -654.132,Z 1277.405,A 0.000,B 0.000,C 90.000,E1 108.906} C_DIS
LIN {X 0.237,Y -657.758,Z 1277.401,A 0.000,B 0.000,C 90.000,E1 108.127} C_DIS
LIN {X 0.106,Y -661.081,Z 1277.397,A 0.000,B 0.000,C 90.000,E1 107.402} C_DIS
LIN {X 0.001,Y -664.094,Z 1277.393,A 0.000,B 0.000,C 90.000,E1 106.677} C_DIS
LIN {X -0.181,Y -665.902,Z 1277.390,A 0.000,B 0.000,C 90.000,E1 106.205} C_DIS
LIN {X -0.247,Y -668.193,Z 1277.386,A 0.000,B 0.000,C 90.000,E1 105.481} C_DIS
LIN {X 0.247,Y -669.544,Z 1277.383,A 0.000,B 0.000,C 90.000,E1 104.954} C_DIS
LIN {X 0.106,Y -670.647,Z 1277.380,A 0.000,B 0.000,C 90.000,E1 104.481} C_DIS
LIN {X -0.090,Y -671.906,Z 1277.376,A 0.000,B 0.000,C 90.000,E1 103.772} C_DIS
LIN {X -0.216,Y -672.557,Z 1277.374,A 0.000,B 0.000,C 90.000,E1 103.300} C_DIS
LIN {X 0.259,Y -673.071,Z 1277.370,A 0.000,B 0.000,C 90.000,E1 102.535} C_DIS
LIN {X 0.140,Y -673.230,Z 1277.367,A 0.000,B 0.000,C 90.000,E1 102.063} C_DIS
LIN {X -0.177,Y -673.046,Z 1277.363,A 0.000,B 0.000,C 90.000,E1 101.366} C_DIS
LIN {X 0.297,Y -672.422,Z 1277.359,A 0.000,B 0.000,C 90.000,E1 100.602} C_DIS
LIN {X 0.232,Y -672.148,Z 1277.358,A 0.000,B 0.000,C 90.000,E1 100.366} C_DIS
LIN {X -0.022,Y -671.304,Z 1277.355,A 0.000,B 0.000,C 90.000,E1 99.905} C_DIS
LIN {X -0.166,Y -670.239,Z 1277.352,A 0.000,B 0.000,C 90.000,E1 99.434} C_DIS
LIN {X 0.234,Y -668.891,Z 1277.350,A 0.000,B 0.000,C 90.000,E1 98.916} C_DIS
LIN {X -0.032,Y -667.159,Z 1277.347,A 0.000,B 0.000,C 90.000,E1 98.454} C_DIS
LIN {X -0.120,Y -666.243,Z 1277.346,A 0.000,B 0.000,C 90.000,E1 98.219} C_DIS
LIN {X 0.164,Y -663.476,Z 1277.342,A 0.000,B 0.000,C 90.000,E1 97.587} C_DIS
LIN {X -0.133,Y -660.877,Z 1277.340,A 0.000,B 0.000,C 90.000,E1 97.125} C_DIS
LIN {X 0.209,Y -657.977,Z 1277.337,A 0.000,B 0.000,C 90.000,E1 96.606} C_DIS
LIN {X -0.155,Y -653.823,Z 1277.333,A 0.000,B 0.000,C 90.000,E1 96.024} C_DIS
LIN {X 0.022,Y -649.140,Z 1277.330,A 0.000,B 0.000,C 90.000,E1 95.391} C_DIS
